KUKA KRL program: EPS_2_25252_PD3_A_20250910061716.src

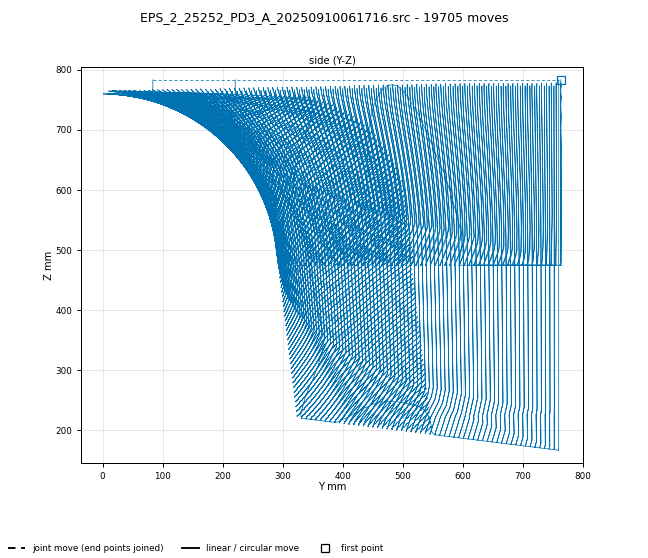
[picture p0: tool path of EPS_2_25252_PD3_A_20250910061716.src, 19705 of 19707 moves have a stored position in this frame; points joined in program order, loops and branches not executed]
&ACCESS RVP
&REL 4
&COMMENT QRS 19112012
&PARAM EDITMASK = *
DEF PART()
EXT BAS (BAS_COMMAND :IN,REAL :IN )
INT I
BAS (#INITMOV,0 )

;KUKA QRS Post kuka4.cps  Date:22-06-2017 !

File_ID=2831

QRS_PRE_INIT()

;Init var - Until changes are made in qrs_pre_init
Outlet_Square_prg=0
Inlet_1_Square_prg=0
Inlet_2_Square_prg=0
Inlet_3_Square_prg=0
Inlet_4_Square_prg=0
Inlet_5_Square_prg=0

Outlet_1={X 0.000, Y 612.000, Z 507.000, B 0.000, E1 0.000 }
Inlet_1={X 0.000, Y 651.000, Z 482.000, B 0.000, E1 180.000 }
Outlet_1_type=533
Inlet_1_type=0
;QRS#1=Sidecore dimensions
;QRS#2=525-21" Concrete
;QRS#3=DeadEnd 533
;QRS#4=
;QRS#5=
;QRS#6=
;QRS#7=
;QRS#8=
;QRS#9=S306-32
;QRS#10=

;QRS#11=
;QRS#12=
;QRS#13=
;QRS#14=
;QRS#15=
;QRS#16=1524x152x1219 4'
;QRS#17=EPS Height
;QRS#18=773,5
;QRS#19=*
;QRS#20= UPDATED VERSION 22-06-2017
;QRS#21=*
Outlet_Square=0350
Inlet_1_Square=00
Inlet_2_Square=0
Inlet_3_Square=0
Inlet_4_Square=0
Inlet_5_Square=0
Mill_Square=1
Outlet_Square_Prg=263
Inlet_1_Square_prg=0

QRS_INIT()

$ADVANCE=5

; T1
PTP {E1 176.574,E2 176.574}
PTP {X 0,Y 763.362,A -85,B 0,C 180,E1 176.574,E2 176.574,E3 0,E4 0,E5 0,E6 0}
QRS_SPEED_INIT()
LIN {X 0,Y 763.362,Z 783.5,A -85,B 0,C 180,E1 176.574,E2 176.574,E3 0,E4 0,E5 0,E6 0} C_VEL
LIN {X 0,Y 763.362,Z 476.78,A -85,B 0,C 180,E1 176.574,E2 176.574} C_VEL
LIN {X 0,Y 763.472,Z 474.78,A -85,B 0,C 180,E1 176.723,E2 176.723} C_VEL
LIN {X 0,Y 763.845,Z 474.78,A -85,B 0,C 180,E1 177.187,E2 177.187} C_VEL
LIN {X 0,Y 763.843,Z 474.78,A -85,B 0,C 180,E1 184.692,E2 184.692} C_VEL
LIN {X 0,Y 763.78,Z 474.78,A -85,B 0,C 180,E1 192.281,E2 192.281} C_VEL
LIN {X 0,Y 763.758,Z 474.78,A -85,B 0,C 180,E1 200.097,E2 200.097} C_VEL
LIN {X 0,Y 763.767,Z 474.78,A -85,B 0,C 180,E1 208.327,E2 208.327} C_VEL
LIN {X 0,Y 762.36,Z 474.78,A -85,B 0,C 180,E1 210.542,E2 210.542} C_VEL
LIN {X 0,Y 762.677,Z 474.78,A -85,B 0,C 180,E1 214.995,E2 214.995} C_VEL
LIN {X 0,Y 763.686,Z 474.78,A -85,B 0,C 180,E1 216.703,E2 216.703} C_VEL
LIN {X 0,Y 763.715,Z 474.78,A -85,B 0,C 180,E1 224.719,E2 224.719} C_VEL
LIN {X 0,Y 763.486,Z 474.78,A -85,B 0,C 180,E1 225.271,E2 225.271} C_VEL
LIN {X 0,Y 762.394,Z 474.78,A -85,B 0,C 180,E1 230.392,E2 230.392} C_VEL
LIN {X 0,Y 763.76,Z 474.78,A -85,B 0,C 180,E1 232.747,E2 232.747} C_VEL
LIN {X 0,Y 763.715,Z 474.78,A -85,B 0,C 180,E1 239.522,E2 239.522} C_VEL
LIN {X 0,Y 763.84,Z 474.78,A -85,B 0,C 180,E1 246.233,E2 246.233} C_VEL
LIN {X 0,Y 763.363,Z 474.78,A -85,B 0,C 180,E1 246.588,E2 246.588} C_VEL
LIN {X 0,Y 762.066,Z 474.78,A -85,B 0,C 180,E1 246.779,E2 246.779} C_VEL
LIN {X 0,Y 761.546,Z 474.78,A -85,B 0,C 180,E1 246.82,E2 246.82} C_VEL
LIN {X 0,Y 762.022,Z 475.377,A -85,B 0,C 180,E1 246.853,E2 246.853} C_VEL
LIN {X 0,Y 763.177,Z 477.146,A -85,B 0,C 180,E1 246.908,E2 246.908} C_VEL
LIN {X 0,Y 763.405,Z 477.716,A -85,B 0,C 180,E1 246.921,E2 246.921} C_VEL
LIN {X 0,Y 763.579,Z 479.406,A -85,B 0,C 180,E1 246.944,E2 246.944} C_VEL
LIN {X 0,Y 763.624,Z 506.616,A -85,B 0,C 180,E1 247.217,E2 247.217} C_VEL
LIN {X 0,Y 763.846,Z 526.018,A -85,B 0,C 180,E1 247.432,E2 247.432} C_VEL
LIN {X 0,Y 763.826,Z 535.654,A -85,B 0,C 180,E1 247.561,E2 247.561} C_VEL
LIN {X 0,Y 763.83,Z 546.762,A -85,B 0,C 180,E1 247.743,E2 247.743} C_VEL
LIN {X 0,Y 763.845,Z 560.557,A -85,B 0,C 180,E1 248.022,E2 248.022} C_VEL
LIN {X 0,Y 763.631,Z 572.226,A -85,B 0,C 180,E1 248.295,E2 248.295} C_VEL
LIN {X 0,Y 763.801,Z 585.949,A -85,B 0,C 180,E1 248.684,E2 248.684} C_VEL
LIN {X 0,Y 763.765,Z 598.566,A -85,B 0,C 180,E1 249.09,E2 249.09} C_VEL
LIN {X 0,Y 763.802,Z 611.561,A -85,B 0,C 180,E1 249.567,E2 249.567} C_VEL
LIN {X 0,Y 763.764,Z 623.559,A -85,B 0,C 180,E1 250.059,E2 250.059} C_VEL
LIN {X 0,Y 763.75,Z 634.569,A -85,B 0,C 180,E1 250.559,E2 250.559} C_VEL
LIN {X 0,Y 763.602,Z 646.52,A -85,B 0,C 180,E1 251.157,E2 251.157} C_VEL
LIN {X 0,Y 763.564,Z 657.079,A -85,B 0,C 180,E1 251.739,E2 251.739} C_VEL
LIN {X 0,Y 763.701,Z 667.628,A -85,B 0,C 180,E1 252.381,E2 252.381} C_VEL
LIN {X 0,Y 763.805,Z 676.976,A -85,B 0,C 180,E1 252.997,E2 252.997} C_VEL
LIN {X 0,Y 763.623,Z 687.198,A -85,B 0,C 180,E1 253.726,E2 253.726} C_VEL
LIN {X 0,Y 763.342,Z 695.759,A -85,B 0,C 180,E1 254.386,E2 254.386} C_VEL
LIN {X 0,Y 763.22,Z 704.692,A -85,B 0,C 180,E1 255.141,E2 255.141} C_VEL
LIN {X 0,Y 763.436,Z 713.229,A -85,B 0,C 180,E1 255.933,E2 255.933} C_VEL
LIN {X 0,Y 763.734,Z 720.481,A -85,B 0,C 180,E1 256.663,E2 256.663} C_VEL
LIN {X 0,Y 763.713,Z 726.434,A -85,B 0,C 180,E1 257.312,E2 257.312} C_VEL
LIN {X 0,Y 763.274,Z 733.979,A -85,B 0,C 180,E1 258.192,E2 258.192} C_VEL
LIN {X 0,Y 763.073,Z 741.325,A -85,B 0,C 180,E1 259.146,E2 259.146} C_VEL
LIN {X 0,Y 763.305,Z 747.875,A -85,B 0,C 180,E1 260.102,E2 260.102} C_VEL
LIN {X 0,Y 763.778,Z 753.687,A -85,B 0,C 180,E1 261.059,E2 261.059} C_VEL
LIN {X 0,Y 763.865,Z 755,A -85,B 0,C 180,E1 261.297,E2 261.297} C_VEL
LIN {X 0,Y 763.317,Z 759.964,A -85,B 0,C 180,E1 262.238,E2 262.238} C_VEL
LIN {X 0,Y 762.989,Z 763.277,A -85,B 0,C 180,E1 262.945,E2 262.945} C_VEL
LIN {X 0,Y 762.889,Z 767.126,A -85,B 0,C 180,E1 263.888,E2 263.888} C_VEL
LIN {X 0,Y 763.222,Z 770.376,A -85,B 0,C 180,E1 264.834,E2 264.834} C_VEL
LIN {X 0,Y 763.816,Z 773.348,A -85,B 0,C 180,E1 265.894,E2 265.894} C_VEL
LIN {X 0,Y 763.592,Z 774.667,A -85,B 0,C 180,E1 266.478,E2 266.478} C_VEL
LIN {X 0,Y 763.145,Z 776.072,A -85,B 0,C 180,E1 267.184,E2 267.184} C_VEL
LIN {X 0,Y 762.829,Z 777.16,A -85,B 0,C 180,E1 267.91,E2 267.91} C_VEL
LIN {X 0,Y 762.834,Z 778.22,A -85,B 0,C 180,E1 269.061,E2 269.061} C_VEL
LIN {X 0,Y 763.862,Z 778.174,A -85,B 0,C 180,E1 270.937,E2 270.937} C_VEL
LIN {X 0,Y 763.613,Z 777.551,A -85,B 0,C 180,E1 271.688,E2 271.688} C_VEL
LIN {X 0,Y 763.495,Z 776.058,A -85,B 0,C 180,E1 272.814,E2 272.814} C_VEL
LIN {X 0,Y 763.659,Z 774.541,A -85,B 0,C 180,E1 273.58,E2 273.58} C_VEL
LIN {X 0,Y 763.841,Z 773.267,A -85,B 0,C 180,E1 274.135,E2 274.135} C_VEL
LIN {X 0,Y 763.624,Z 771.764,A -85,B 0,C 180,E1 274.693,E2 274.693} C_VEL
LIN {X 0,Y 763.089,Z 768.798,A -85,B 0,C 180,E1 275.638,E2 275.638} C_VEL
LIN {X 0,Y 762.918,Z 767.126,A -85,B 0,C 180,E1 276.111,E2 276.111} C_VEL
LIN {X 0,Y 762.9,Z 763.277,A -85,B 0,C 180,E1 277.056,E2 277.056} C_VEL
LIN {X 0,Y 763.306,Z 758.808,A -85,B 0,C 180,E1 277.998,E2 277.998} C_VEL
LIN {X 0,Y 763.85,Z 753.687,A -85,B 0,C 180,E1 278.94,E2 278.94} C_VEL
LIN {X 0,Y 763.421,Z 747.875,A -85,B 0,C 180,E1 279.896,E2 279.896} C_VEL
LIN {X 0,Y 763.086,Z 741.325,A -85,B 0,C 180,E1 280.854,E2 280.854} C_VEL
LIN {X 0,Y 763.195,Z 733.979,A -85,B 0,C 180,E1 281.809,E2 281.809} C_VEL
LIN {X 0,Y 763.537,Z 727.593,A -85,B 0,C 180,E1 282.565,E2 282.565} C_VEL
LIN {X 0,Y 763.83,Z 720.63,A -85,B 0,C 180,E1 283.319,E2 283.319} C_VEL
LIN {X 0,Y 763.441,Z 710.557,A -85,B 0,C 180,E1 284.319,E2 284.319} C_VEL
LIN {X 0,Y 763.239,Z 702.208,A -85,B 0,C 180,E1 285.074,E2 285.074} C_VEL
LIN {X 0,Y 763.3,Z 694.06,A -85,B 0,C 180,E1 285.751,E2 285.751} C_VEL
LIN {X 0,Y 763.618,Z 683.872,A -85,B 0,C 180,E1 286.518,E2 286.518} C_VEL
LIN {X 0,Y 763.769,Z 675.166,A -85,B 0,C 180,E1 287.127,E2 287.127} C_VEL
LIN {X 0,Y 763.695,Z 663.646,A -85,B 0,C 180,E1 287.866,E2 287.866} C_VEL
LIN {X 0,Y 763.565,Z 654.622,A -85,B 0,C 180,E1 288.403,E2 288.403} C_VEL
LIN {X 0,Y 763.593,Z 642.535,A -85,B 0,C 180,E1 289.05,E2 289.05} C_VEL
LIN {X 0,Y 763.737,Z 630.359,A -85,B 0,C 180,E1 289.637,E2 289.637} C_VEL
LIN {X 0,Y 763.711,Z 620.01,A -85,B 0,C 180,E1 290.096,E2 290.096} C_VEL
LIN {X 0,Y 763.808,Z 608.143,A -85,B 0,C 180,E1 290.566,E2 290.566} C_VEL
LIN {X 0,Y 763.711,Z 594.677,A -85,B 0,C 180,E1 291.043,E2 291.043} C_VEL
LIN {X 0,Y 763.729,Z 582.345,A -85,B 0,C 180,E1 291.425,E2 291.425} C_VEL
LIN {X 0,Y 763.792,Z 568.153,A -85,B 0,C 180,E1 291.801,E2 291.801} C_VEL
LIN {X 0,Y 763.649,Z 556.327,A -85,B 0,C 180,E1 292.077,E2 292.077} C_VEL
LIN {X 0,Y 763.845,Z 541.803,A -85,B 0,C 180,E1 292.342,E2 292.342} C_VEL
LIN {X 0,Y 763.851,Z 529.818,A -85,B 0,C 180,E1 292.523,E2 292.523} C_VEL
LIN {X 0,Y 763.83,Z 511.799,A -85,B 0,C 180,E1 292.724,E2 292.724} C_VEL
LIN {X 0,Y 763.611,Z 481.566,A -85,B 0,C 180,E1 293.034,E2 293.034} C_VEL
LIN {X 0,Y 763.361,Z 477.535,A -85,B 0,C 180,E1 293.082,E2 293.082} C_VEL
LIN {X 0,Y 762.558,Z 474.78,A -85,B 0,C 180,E1 293.148,E2 293.148} C_VEL
LIN {X 0,Y 763.365,Z 474.78,A -85,B 0,C 180,E1 293.244,E2 293.244} C_VEL
LIN {X 0,Y 763.723,Z 474.78,A -85,B 0,C 180,E1 293.756,E2 293.756} C_VEL
LIN {X 0,Y 763.844,Z 474.78,A -85,B 0,C 180,E1 298.32,E2 298.32} C_VEL
LIN {X 0,Y 763.726,Z 474.78,A -85,B 0,C 180,E1 304.935,E2 304.935} C_VEL
LIN {X 0,Y 762.49,Z 474.78,A -85,B 0,C 180,E1 307.326,E2 307.326} C_VEL
LIN {X 0,Y 763.687,Z 474.78,A -85,B 0,C 180,E1 312.132,E2 312.132} C_VEL
LIN {X 0,Y 763.532,Z 474.78,A -85,B 0,C 180,E1 312.563,E2 312.563} C_VEL
LIN {X 0,Y 763.766,Z 474.78,A -85,B 0,C 180,E1 320.258,E2 320.258} C_VEL
LIN {X 0,Y 763.66,Z 474.78,A -85,B 0,C 180,E1 326.563,E2 326.563} C_VEL
LIN {X 0,Y 763.416,Z 474.78,A -85,B 0,C 180,E1 327.302,E2 327.302} C_VEL
LIN {X 0,Y 763.767,Z 474.78,A -85,B 0,C 180,E1 333.782,E2 333.782} C_VEL
LIN {X 0,Y 763.76,Z 474.78,A -85,B 0,C 180,E1 341.887,E2 341.887} C_VEL
LIN {X 0,Y 763.788,Z 474.78,A -85,B 0,C 180,E1 349.631,E2 349.631} C_VEL
LIN {X 0,Y 763.844,Z 474.78,A -85,B 0,C 180,E1 357.187,E2 357.187} C_VEL
LIN {X 0,Y 763.835,Z 474.78,A -85,B 0,C 180,E1 364.692,E2 364.692} C_VEL
LIN {X 0,Y 763.773,Z 474.78,A -85,B 0,C 180,E1 372.281,E2 372.281} C_VEL
LIN {X 0,Y 763.757,Z 474.78,A -85,B 0,C 180,E1 380.097,E2 380.097} C_VEL
LIN {X 0,Y 763.776,Z 474.78,A -85,B 0,C 180,E1 388.327,E2 388.327} C_VEL
LIN {X 0,Y 763.753,Z 474.78,A -85,B 0,C 180,E1 394.938,E2 394.938} C_VEL
LIN {X 0,Y 762.455,Z 474.78,A -85,B 0,C 180,E1 399.735,E2 399.735} C_VEL
LIN {X 0,Y 763.747,Z 474.78,A -85,B 0,C 180,E1 402.135,E2 402.135} C_VEL
LIN {X 0,Y 763.573,Z 474.78,A -85,B 0,C 180,E1 402.574,E2 402.574} C_VEL
LIN {X 0,Y 763.844,Z 474.78,A -85,B 0,C 180,E1 410.26,E2 410.26} C_VEL
LIN {X 0,Y 763.674,Z 474.78,A -85,B 0,C 180,E1 416.573,E2 416.573} C_VEL
LIN {X 0,Y 763.421,Z 474.78,A -85,B 0,C 180,E1 417.307,E2 417.307} C_VEL
LIN {X 0,Y 763.747,Z 474.78,A -85,B 0,C 180,E1 423.785,E2 423.785} C_VEL
LIN {X 0,Y 763.796,Z 474.78,A -85,B 0,C 180,E1 431.89,E2 431.89} C_VEL
LIN {X 0,Y 763.784,Z 474.78,A -85,B 0,C 180,E1 439.633,E2 439.633} C_VEL
LIN {X 0,Y 763.772,Z 474.78,A -85,B 0,C 180,E1 447.187,E2 447.187} C_VEL
LIN {X 0,Y 763.776,Z 474.78,A -85,B 0,C 180,E1 454.692,E2 454.692} C_VEL
LIN {X 0,Y 763.786,Z 474.78,A -85,B 0,C 180,E1 462.279,E2 462.279} C_VEL
LIN {X 0,Y 763.785,Z 474.78,A -85,B 0,C 180,E1 470.094,E2 470.094} C_VEL
LIN {X 0,Y 763.728,Z 474.78,A -85,B 0,C 180,E1 478.325,E2 478.325} C_VEL
LIN {X 0,Y 761.89,Z 474.78,A -85,B 0,C 180,E1 482.767,E2 482.767} C_VEL
LIN {X 0,Y 762.616,Z 474.78,A -85,B 0,C 180,E1 484.993,E2 484.993} C_VEL
LIN {X 0,Y 763.623,Z 474.78,A -85,B 0,C 180,E1 486.687,E2 486.687} C_VEL
LIN {X 0,Y 763.669,Z 474.78,A -85,B 0,C 180,E1 494.715,E2 494.715} C_VEL
LIN {X 0,Y 763.456,Z 474.78,A -85,B 0,C 180,E1 495.262,E2 495.262} C_VEL
LIN {X 0,Y 762.344,Z 474.78,A -85,B 0,C 180,E1 500.387,E2 500.387} C_VEL
LIN {X 0,Y 763.704,Z 474.78,A -85,B 0,C 180,E1 502.738,E2 502.738} C_VEL
LIN {X 0,Y 763.588,Z 474.78,A -85,B 0,C 180,E1 510.146,E2 510.146} C_VEL
LIN {X 0,Y 762.882,Z 474.78,A -85,B 0,C 180,E1 511.637,E2 511.637} C_VEL
LIN {X 0,Y 763.752,Z 474.78,A -85,B 0,C 180,E1 517.893,E2 517.893} C_VEL
LIN {X 0,Y 763.489,Z 474.78,A -85,B 0,C 180,E1 524.93,E2 524.93} C_VEL
LIN {X 0,Y 763.662,Z 474.78,A -85,B 0,C 180,E1 525.79,E2 525.79} C_VEL
LIN {X 0,Y 763.795,Z 474.78,A -85,B 0,C 180,E1 529.631,E2 529.631} C_VEL
LIN {X 0,Y 763.472,Z 474.78,A -85,B 0,C 180,E1 536.723,E2 536.723} C_VEL
LIN {X 0,Y 754.509,Z 474.78,A -85,B 0,C 180,E1 539.325,E2 539.325} C_VEL
LIN {X 0,Y 754.692,Z 474.78,A -85,B 0,C 180,E1 546.383,E2 546.383} C_VEL
LIN {X 0,Y 754.905,Z 474.78,A -85,B 0,C 180,E1 553.399,E2 553.399} C_VEL
LIN {X 0,Y 755.041,Z 474.78,A -85,B 0,C 180,E1 560.942,E2 560.942} C_VEL
LIN {X 0,Y 754.868,Z 474.78,A -85,B 0,C 180,E1 569.54,E2 569.54} C_VEL
LIN {X 0,Y 754.766,Z 474.78,A -85,B 0,C 180,E1 577.858,E2 577.858} C_VEL
LIN {X 0,Y 754.887,Z 474.78,A -85,B 0,C 180,E1 586.126,E2 586.126} C_VEL
LIN {X 0,Y 755.149,Z 474.78,A -85,B 0,C 180,E1 593.671,E2 593.671} C_VEL
LIN {X 0,Y 754.823,Z 474.78,A -85,B 0,C 180,E1 601.041,E2 601.041} C_VEL
LIN {X 0,Y 754.166,Z 474.78,A -85,B 0,C 180,E1 606.591,E2 606.591} C_VEL
LIN {X 0,Y 756.39,Z 562.55,A -85,B 0,C 180,E1 607.841,E2 607.841} C_VEL
LIN {X 0,Y 756.168,Z 623.267,A -85,B 0,C 180,E1 609.837,E2 609.837} C_VEL
LIN {X 0,Y 756.007,Z 677.473,A -85,B 0,C 180,E1 612.852,E2 612.852} C_VEL
LIN {X 0,Y 755.802,Z 721.742,A -85,B 0,C 180,E1 616.659,E2 616.659} C_VEL
LIN {X 0,Y 755.794,Z 754.21,A -85,B 0,C 180,E1 621.054,E2 621.054} C_VEL
LIN {X 0,Y 755.805,Z 773.709,A -85,B 0,C 180,E1 625.973,E2 625.973} C_VEL
LIN {X 0,Y 755.615,Z 778.34,A -85,B 0,C 180,E1 630.575,E2 630.575} C_VEL
LIN {X 0,Y 755.326,Z 770.506,A -85,B 0,C 180,E1 635.184,E2 635.184} C_VEL
LIN {X 0,Y 755.484,Z 748.988,A -85,B 0,C 180,E1 639.824,E2 639.824} C_VEL
LIN {X 0,Y 755.589,Z 713.063,A -85,B 0,C 180,E1 644.233,E2 644.233} C_VEL
LIN {X 0,Y 755.936,Z 664.27,A -85,B 0,C 180,E1 648.018,E2 648.018} C_VEL
LIN {X 0,Y 756.249,Z 606.531,A -85,B 0,C 180,E1 650.84,E2 650.84} C_VEL
LIN {X 0,Y 756.434,Z 543.515,A -85,B 0,C 180,E1 652.545,E2 652.545} C_VEL
LIN {X 0,Y 755.352,Z 474.78,A -85,B 0,C 180,E1 653.409,E2 653.409} C_VEL
LIN {X 0,Y 755.098,Z 474.78,A -85,B 0,C 180,E1 659.475,E2 659.475} C_VEL
LIN {X 0,Y 754.862,Z 474.78,A -85,B 0,C 180,E1 666.345,E2 666.345} C_VEL
LIN {X 0,Y 755.342,Z 474.78,A -85,B 0,C 180,E1 672.798,E2 672.798} C_VEL
LIN {X 0,Y 755.448,Z 474.78,A -85,B 0,C 180,E1 680.711,E2 680.711} C_VEL
LIN {X 0,Y 755.103,Z 474.78,A -85,B 0,C 180,E1 687.787,E2 687.787} C_VEL
LIN {X 0,Y 755.266,Z 474.78,A -85,B 0,C 180,E1 694.373,E2 694.373} C_VEL
LIN {X 0,Y 754.891,Z 474.78,A -85,B 0,C 180,E1 703.021,E2 703.021} C_VEL
LIN {X 0,Y 755.374,Z 474.78,A -85,B 0,C 180,E1 710.135,E2 710.135} C_VEL
LIN {X 0,Y 755.05,Z 474.78,A -85,B 0,C 180,E1 718.238,E2 718.238} C_VEL
LIN {X 0,Y 754.845,Z 474.78,A -85,B 0,C 180,E1 726.036,E2 726.036} C_VEL
LIN {X 0,Y 754.937,Z 474.78,A -85,B 0,C 180,E1 733.327,E2 733.327} C_VEL
LIN {X 0,Y 755.046,Z 474.78,A -85,B 0,C 180,E1 740.943,E2 740.943} C_VEL
LIN {X 0,Y 755.058,Z 474.78,A -85,B 0,C 180,E1 749.452,E2 749.452} C_VEL
LIN {X 0,Y 754.823,Z 474.78,A -85,B 0,C 180,E1 756.324,E2 756.324} C_VEL
LIN {X 0,Y 755.323,Z 474.78,A -85,B 0,C 180,E1 762.877,E2 762.877} C_VEL
LIN {X 0,Y 755.472,Z 474.78,A -85,B 0,C 180,E1 770.779,E2 770.779} C_VEL
LIN {X 0,Y 755.079,Z 474.78,A -85,B 0,C 180,E1 777.844,E2 777.844} C_VEL
LIN {X 0,Y 755.203,Z 474.78,A -85,B 0,C 180,E1 784.423,E2 784.423} C_VEL
LIN {X 0,Y 754.891,Z 474.78,A -85,B 0,C 180,E1 793.065,E2 793.065} C_VEL
LIN {X 0,Y 755.331,Z 474.78,A -85,B 0,C 180,E1 800.174,E2 800.174} C_VEL
LIN {X 0,Y 754.958,Z 474.78,A -85,B 0,C 180,E1 808.273,E2 808.273} C_VEL
LIN {X 0,Y 754.788,Z 474.78,A -85,B 0,C 180,E1 816.063,E2 816.063} C_VEL
LIN {X 0,Y 754.932,Z 474.78,A -85,B 0,C 180,E1 823.357,E2 823.357} C_VEL
LIN {X 0,Y 755.023,Z 474.78,A -85,B 0,C 180,E1 830.963,E2 830.963} C_VEL
LIN {X 0,Y 754.794,Z 474.78,A -85,B 0,C 180,E1 839.488,E2 839.488} C_VEL
LIN {X 0,Y 754.728,Z 474.78,A -85,B 0,C 180,E1 847.795,E2 847.795} C_VEL
LIN {X 0,Y 754.835,Z 474.78,A -85,B 0,C 180,E1 856.144,E2 856.144} C_VEL
LIN {X 0,Y 754.97,Z 474.78,A -85,B 0,C 180,E1 863.684,E2 863.684} C_VEL
LIN {X 0,Y 754.771,Z 474.78,A -85,B 0,C 180,E1 871.85,E2 871.85} C_VEL
LIN {X 0,Y 754.717,Z 474.78,A -85,B 0,C 180,E1 879.439,E2 879.439} C_VEL
LIN {X 0,Y 755.375,Z 474.78,A -85,B 0,C 180,E1 886.827,E2 886.827} C_VEL
LIN {X 0,Y 754.178,Z 474.78,A -85,B 0,C 180,E1 893.682,E2 893.682} C_VEL
LIN {X 0,Y 755.031,Z 474.78,A -85,B 0,C 180,E1 898.307,E2 898.307} C_VEL
LIN {X 0,Y 754.509,Z 474.78,A -85,B 0,C 180,E1 899.325,E2 899.325} C_VEL
LIN {X 0,Y 746.359,Z 474.78,A -85,B 0,C 180,E1 901.958,E2 901.958} C_VEL
LIN {X 0,Y 746.234,Z 474.78,A -85,B 0,C 180,E1 907.629,E2 907.629} C_VEL
LIN {X 0,Y 746.807,Z 474.78,A -85,B 0,C 180,E1 913.547,E2 913.547} C_VEL
LIN {X 0,Y 747.111,Z 474.78,A -85,B 0,C 180,E1 920.854,E2 920.854} C_VEL
LIN {X 0,Y 747.442,Z 474.78,A -85,B 0,C 180,E1 928.531,E2 928.531} C_VEL
LIN {X 0,Y 747.23,Z 474.78,A -85,B 0,C 180,E1 936.841,E2 936.841} C_VEL
LIN {X 0,Y 747.247,Z 474.78,A -85,B 0,C 180,E1 945.561,E2 945.561} C_VEL
LIN {X 0,Y 747.244,Z 474.78,A -85,B 0,C 180,E1 953.381,E2 953.381} C_VEL
LIN {X 0,Y 747.137,Z 474.78,A -85,B 0,C 180,E1 960.179,E2 960.179} C_VEL
LIN {X 0,Y 746.841,Z 475.472,A -85,B 0,C 180,E1 966.356,E2 966.356} C_VEL
LIN {X 0,Y 748.969,Z 562.274,A -85,B 0,C 180,E1 967.603,E2 967.603} C_VEL
LIN {X 0,Y 748.558,Z 623.266,A -85,B 0,C 180,E1 969.623,E2 969.623} C_VEL
LIN {X 0,Y 748.205,Z 677.856,A -85,B 0,C 180,E1 972.695,E2 972.695} C_VEL
LIN {X 0,Y 747.901,Z 723.112,A -85,B 0,C 180,E1 976.669,E2 976.669} C_VEL
LIN {X 0,Y 747.831,Z 755.753,A -85,B 0,C 180,E1 981.252,E2 981.252} C_VEL
LIN {X 0,Y 747.79,Z 773.708,A -85,B 0,C 180,E1 985.93,E2 985.93} C_VEL
LIN {X 0,Y 747.609,Z 778.34,A -85,B 0,C 180,E1 990.581,E2 990.581} C_VEL
LIN {X 0,Y 747.293,Z 770.508,A -85,B 0,C 180,E1 995.239,E2 995.239} C_VEL
LIN {X 0,Y 747.479,Z 748.984,A -85,B 0,C 180,E1 999.93,E2 999.93} C_VEL
LIN {X 0,Y 747.658,Z 713.056,A -85,B 0,C 180,E1 1004.387,E2 1004.387} C_VEL
LIN {X 0,Y 748.186,Z 664.011,A -85,B 0,C 180,E1 1008.227,E2 1008.227} C_VEL
LIN {X 0,Y 748.669,Z 606.542,A -85,B 0,C 180,E1 1011.061,E2 1011.061} C_VEL
LIN {X 0,Y 749.031,Z 544.136,A -85,B 0,C 180,E1 1012.769,E2 1012.769} C_VEL
LIN {X 0,Y 747.589,Z 474.78,A -85,B 0,C 180,E1 1013.718,E2 1013.718} C_VEL
LIN {X 0,Y 746.777,Z 474.78,A -85,B 0,C 180,E1 1020.223,E2 1020.223} C_VEL
LIN {X 0,Y 746.686,Z 474.78,A -85,B 0,C 180,E1 1026.808,E2 1026.808} C_VEL
LIN {X 0,Y 746.669,Z 474.78,A -85,B 0,C 180,E1 1033.783,E2 1033.783} C_VEL
LIN {X 0,Y 746.949,Z 474.78,A -85,B 0,C 180,E1 1041.674,E2 1041.674} C_VEL
LIN {X 0,Y 746.669,Z 474.78,A -85,B 0,C 180,E1 1048.751,E2 1048.751} C_VEL
LIN {X 0,Y 746.571,Z 474.78,A -85,B 0,C 180,E1 1055.341,E2 1055.341} C_VEL
LIN {X 0,Y 747.02,Z 474.78,A -85,B 0,C 180,E1 1062.836,E2 1062.836} C_VEL
LIN {X 0,Y 746.698,Z 474.78,A -85,B 0,C 180,E1 1071.199,E2 1071.199} C_VEL
LIN {X 0,Y 747.053,Z 474.78,A -85,B 0,C 180,E1 1078.219,E2 1078.219} C_VEL
LIN {X 0,Y 747.412,Z 474.78,A -85,B 0,C 180,E1 1085.206,E2 1085.206} C_VEL
LIN {X 0,Y 746.837,Z 474.78,A -85,B 0,C 180,E1 1093.475,E2 1093.475} C_VEL
LIN {X 0,Y 747.157,Z 474.78,A -85,B 0,C 180,E1 1100.778,E2 1100.778} C_VEL
LIN {X 0,Y 747.444,Z 474.78,A -85,B 0,C 180,E1 1108.451,E2 1108.451} C_VEL
LIN {X 0,Y 747.436,Z 474.78,A -85,B 0,C 180,E1 1115.304,E2 1115.304} C_VEL
LIN {X 0,Y 747.357,Z 474.78,A -85,B 0,C 180,E1 1122.803,E2 1122.803} C_VEL
LIN {X 0,Y 746.965,Z 474.78,A -85,B 0,C 180,E1 1131.742,E2 1131.742} C_VEL
LIN {X 0,Y 746.637,Z 474.78,A -85,B 0,C 180,E1 1138.807,E2 1138.807} C_VEL
LIN {X 0,Y 746.534,Z 474.78,A -85,B 0,C 180,E1 1145.391,E2 1145.391} C_VEL
LIN {X 0,Y 747.005,Z 474.78,A -85,B 0,C 180,E1 1152.881,E2 1152.881} C_VEL
LIN {X 0,Y 747.314,Z 474.78,A -85,B 0,C 180,E1 1160.068,E2 1160.068} C_VEL
LIN {X 0,Y 746.961,Z 474.78,A -85,B 0,C 180,E1 1168.255,E2 1168.255} C_VEL
LIN {X 0,Y 747.336,Z 474.78,A -85,B 0,C 180,E1 1175.239,E2 1175.239} C_VEL
LIN {X 0,Y 746.833,Z 474.78,A -85,B 0,C 180,E1 1183.504,E2 1183.504} C_VEL
LIN {X 0,Y 747.137,Z 474.78,A -85,B 0,C 180,E1 1190.806,E2 1190.806} C_VEL
LIN {X 0,Y 747.373,Z 474.78,A -85,B 0,C 180,E1 1198.479,E2 1198.479} C_VEL
LIN {X 0,Y 747.147,Z 474.78,A -85,B 0,C 180,E1 1206.781,E2 1206.781} C_VEL
LIN {X 0,Y 746.84,Z 474.78,A -85,B 0,C 180,E1 1216.124,E2 1216.124} C_VEL
LIN {X 0,Y 747.112,Z 474.78,A -85,B 0,C 180,E1 1223.3,E2 1223.3} C_VEL
LIN {X 0,Y 746.661,Z 474.78,A -85,B 0,C 180,E1 1232.067,E2 1232.067} C_VEL
LIN {X 0,Y 746.852,Z 474.78,A -85,B 0,C 180,E1 1239.213,E2 1239.213} C_VEL
LIN {X 0,Y 747.328,Z 474.78,A -85,B 0,C 180,E1 1247.728,E2 1247.728} C_VEL
LIN {X 0,Y 747.783,Z 474.78,A -85,B 0,C 180,E1 1257.127,E2 1257.127} C_VEL
LIN {X 0,Y 746.359,Z 474.78,A -85,B 0,C 180,E1 1261.958,E2 1261.958} C_VEL
LIN {X 0,Y 739.299,Z 474.78,A -85,B 0,C 180,E1 1264.638,E2 1264.638} C_VEL
LIN {X 0,Y 738.728,Z 474.78,A -85,B 0,C 180,E1 1273.698,E2 1273.698} C_VEL
LIN {X 0,Y 738.919,Z 474.78,A -85,B 0,C 180,E1 1281.097,E2 1281.097} C_VEL
LIN {X 0,Y 738.946,Z 474.78,A -85,B 0,C 180,E1 1289.285,E2 1289.285} C_VEL
LIN {X 0,Y 738.703,Z 474.78,A -85,B 0,C 180,E1 1297.78,E2 1297.78} C_VEL
LIN {X 0,Y 739.312,Z 474.78,A -85,B 0,C 180,E1 1305.123,E2 1305.123} C_VEL
LIN {X 0,Y 738.84,Z 474.78,A -85,B 0,C 180,E1 1314.267,E2 1314.267} C_VEL
LIN {X 0,Y 738.752,Z 474.78,A -85,B 0,C 180,E1 1321.158,E2 1321.158} C_VEL
LIN {X 0,Y 739.506,Z 476.426,A -85,B 0,C 180,E1 1326.116,E2 1326.116} C_VEL
LIN {X 0,Y 741.559,Z 562.703,A -85,B 0,C 180,E1 1327.377,E2 1327.377} C_VEL
LIN {X 0,Y 740.98,Z 623.251,A -85,B 0,C 180,E1 1329.405,E2 1329.405} C_VEL
LIN {X 0,Y 740.408,Z 678.774,A -85,B 0,C 180,E1 1332.575,E2 1332.575} C_VEL
LIN {X 0,Y 739.988,Z 723.549,A -85,B 0,C 180,E1 1336.573,E2 1336.573} C_VEL
LIN {X 0,Y 739.826,Z 755.755,A -85,B 0,C 180,E1 1341.157,E2 1341.157} C_VEL
LIN {X 0,Y 739.762,Z 773.706,A -85,B 0,C 180,E1 1345.886,E2 1345.886} C_VEL
LIN {X 0,Y 739.603,Z 778.34,A -85,B 0,C 180,E1 1350.587,E2 1350.587} C_VEL
LIN {X 0,Y 739.288,Z 770.51,A -85,B 0,C 180,E1 1355.296,E2 1355.296} C_VEL
LIN {X 0,Y 739.489,Z 748.981,A -85,B 0,C 180,E1 1360.039,E2 1360.039} C_VEL
LIN {X 0,Y 739.734,Z 713.05,A -85,B 0,C 180,E1 1364.544,E2 1364.544} C_VEL
LIN {X 0,Y 740.441,Z 664.852,A -85,B 0,C 180,E1 1368.372,E2 1368.372} C_VEL
LIN {X 0,Y 741.129,Z 606.769,A -85,B 0,C 180,E1 1371.277,E2 1371.277} C_VEL
LIN {X 0,Y 741.675,Z 542.984,A -85,B 0,C 180,E1 1373.027,E2 1373.027} C_VEL
LIN {X 0,Y 739.593,Z 474.78,A -85,B 0,C 180,E1 1373.917,E2 1373.917} C_VEL
LIN {X 0,Y 738.533,Z 474.78,A -85,B 0,C 180,E1 1381.441,E2 1381.441} C_VEL
LIN {X 0,Y 738.412,Z 474.78,A -85,B 0,C 180,E1 1387.658,E2 1387.658} C_VEL
LIN {X 0,Y 738.865,Z 474.78,A -85,B 0,C 180,E1 1393.438,E2 1393.438} C_VEL
LIN {X 0,Y 739.098,Z 474.78,A -85,B 0,C 180,E1 1401.192,E2 1401.192} C_VEL
LIN {X 0,Y 738.801,Z 474.78,A -85,B 0,C 180,E1 1408.413,E2 1408.413} C_VEL
LIN {X 0,Y 738.763,Z 474.78,A -85,B 0,C 180,E1 1415.063,E2 1415.063} C_VEL
LIN {X 0,Y 739.103,Z 474.78,A -85,B 0,C 180,E1 1422.646,E2 1422.646} C_VEL
LIN {X 0,Y 738.736,Z 474.78,A -85,B 0,C 180,E1 1431.104,E2 1431.104} C_VEL
LIN {X 0,Y 739.057,Z 474.78,A -85,B 0,C 180,E1 1438.2,E2 1438.2} C_VEL
LIN {X 0,Y 739.091,Z 474.78,A -85,B 0,C 180,E1 1445.654,E2 1445.654} C_VEL
LIN {X 0,Y 738.764,Z 474.78,A -85,B 0,C 180,E1 1453.625,E2 1453.625} C_VEL
LIN {X 0,Y 738.989,Z 474.78,A -85,B 0,C 180,E1 1461.019,E2 1461.019} C_VEL
LIN {X 0,Y 739.049,Z 474.78,A -85,B 0,C 180,E1 1469.299,E2 1469.299} C_VEL
LIN {X 0,Y 739.064,Z 474.78,A -85,B 0,C 180,E1 1475.855,E2 1475.855} C_VEL
LIN {X 0,Y 738.916,Z 474.78,A -85,B 0,C 180,E1 1483.412,E2 1483.412} C_VEL
LIN {X 0,Y 739.18,Z 474.78,A -85,B 0,C 180,E1 1491.264,E2 1491.264} C_VEL
LIN {X 0,Y 738.751,Z 474.78,A -85,B 0,C 180,E1 1498.436,E2 1498.436} C_VEL
LIN {X 0,Y 738.7,Z 474.78,A -85,B 0,C 180,E1 1505.112,E2 1505.112} C_VEL
LIN {X 0,Y 739.073,Z 474.78,A -85,B 0,C 180,E1 1512.691,E2 1512.691} C_VEL
LIN {X 0,Y 738.739,Z 474.78,A -85,B 0,C 180,E1 1521.144,E2 1521.144} C_VEL
LIN {X 0,Y 738.965,Z 474.78,A -85,B 0,C 180,E1 1528.236,E2 1528.236} C_VEL
LIN {X 0,Y 739.026,Z 474.78,A -85,B 0,C 180,E1 1535.683,E2 1535.683} C_VEL
LIN {X 0,Y 738.761,Z 474.78,A -85,B 0,C 180,E1 1543.654,E2 1543.654} C_VEL
LIN {X 0,Y 738.952,Z 474.78,A -85,B 0,C 180,E1 1551.047,E2 1551.047} C_VEL
LIN {X 0,Y 738.858,Z 474.78,A -85,B 0,C 180,E1 1559.296,E2 1559.296} C_VEL
LIN {X 0,Y 738.618,Z 474.78,A -85,B 0,C 180,E1 1567.794,E2 1567.794} C_VEL
LIN {X 0,Y 739.273,Z 474.78,A -85,B 0,C 180,E1 1575.049,E2 1575.049} C_VEL
LIN {X 0,Y 738.627,Z 474.78,A -85,B 0,C 180,E1 1584.211,E2 1584.211} C_VEL
LIN {X 0,Y 738.924,Z 474.78,A -85,B 0,C 180,E1 1591.19,E2 1591.19} C_VEL
LIN {X 0,Y 738.923,Z 474.78,A -85,B 0,C 180,E1 1599.034,E2 1599.034} C_VEL
LIN {X 0,Y 739.32,Z 474.78,A -85,B 0,C 180,E1 1607.592,E2 1607.592} C_VEL
LIN {X 0,Y 739.742,Z 474.78,A -85,B 0,C 180,E1 1617.096,E2 1617.096} C_VEL
LIN {X 0,Y 739.299,Z 474.78,A -85,B 0,C 180,E1 1624.638,E2 1624.638} C_VEL
LIN {X 0,Y 730.319,Z 474.78,A -85,B 0,C 180,E1 1627.314,E2 1627.314} C_VEL
LIN {X 0,Y 730.642,Z 474.78,A -85,B 0,C 180,E1 1633.853,E2 1633.853} C_VEL
LIN {X 0,Y 730.744,Z 474.78,A -85,B 0,C 180,E1 1641.344,E2 1641.344} C_VEL
LIN {X 0,Y 730.968,Z 474.78,A -85,B 0,C 180,E1 1649.235,E2 1649.235} C_VEL
LIN {X 0,Y 730.687,Z 474.78,A -85,B 0,C 180,E1 1657.819,E2 1657.819} C_VEL
LIN {X 0,Y 730.867,Z 474.78,A -85,B 0,C 180,E1 1665.965,E2 1665.965} C_VEL
LIN {X 0,Y 730.903,Z 474.78,A -85,B 0,C 180,E1 1673.749,E2 1673.749} C_VEL
LIN {X 0,Y 730.898,Z 474.78,A -85,B 0,C 180,E1 1680.818,E2 1680.818} C_VEL
LIN {X 0,Y 731.284,Z 475.314,A -85,B 0,C 180,E1 1685.819,E2 1685.819} C_VEL
LIN {X 0,Y 734.249,Z 506.523,A -85,B 0,C 180,E1 1686.25,E2 1686.25} C_VEL
LIN {X 0,Y 733.85,Z 574.284,A -85,B 0,C 180,E1 1687.426,E2 1687.426} C_VEL
LIN {X 0,Y 733.236,Z 634.845,A -85,B 0,C 180,E1 1689.731,E2 1689.731} C_VEL
LIN {X 0,Y 732.474,Z 686.979,A -85,B 0,C 180,E1 1692.996,E2 1692.996} C_VEL
LIN {X 0,Y 731.936,Z 729.943,A -85,B 0,C 180,E1 1697.171,E2 1697.171} C_VEL
LIN {X 0,Y 731.511,Z 760.235,A -85,B 0,C 180,E1 1701.956,E2 1701.956} C_VEL
LIN {X 0,Y 731.249,Z 776.055,A -85,B 0,C 180,E1 1707.028,E2 1707.028} C_VEL
LIN {X 0,Y 731.632,Z 777.587,A -85,B 0,C 180,E1 1711.782,E2 1711.782} C_VEL
LIN {X 0,Y 730.931,Z 766.48,A -85,B 0,C 180,E1 1716.552,E2 1716.552} C_VEL
LIN {X 0,Y 731.279,Z 743.181,A -85,B 0,C 180,E1 1721.059,E2 1721.059} C_VEL
LIN {X 0,Y 731.827,Z 707.146,A -85,B 0,C 180,E1 1725.279,E2 1725.279} C_VEL
LIN {X 0,Y 732.718,Z 657.863,A -85,B 0,C 180,E1 1729.011,E2 1729.011} C_VEL
LIN {X 0,Y 733.669,Z 599.036,A -85,B 0,C 180,E1 1731.795,E2 1731.795} C_VEL
LIN {X 0,Y 734.348,Z 537.102,A -85,B 0,C 180,E1 1733.37,E2 1733.37} C_VEL
LIN {X 0,Y 732.124,Z 477.807,A -85,B 0,C 180,E1 1734.125,E2 1734.125} C_VEL
LIN {X 0,Y 731.46,Z 474.78,A -85,B 0,C 180,E1 1734.283,E2 1734.283} C_VEL
LIN {X 0,Y 730.682,Z 474.78,A -85,B 0,C 180,E1 1740.563,E2 1740.563} C_VEL
LIN {X 0,Y 730.633,Z 474.78,A -85,B 0,C 180,E1 1746.86,E2 1746.86} C_VEL
LIN {X 0,Y 730.466,Z 474.78,A -85,B 0,C 180,E1 1754.176,E2 1754.176} C_VEL
LIN {X 0,Y 730.796,Z 474.78,A -85,B 0,C 180,E1 1762.188,E2 1762.188} C_VEL
LIN {X 0,Y 730.522,Z 474.78,A -85,B 0,C 180,E1 1769.372,E2 1769.372} C_VEL
LIN {X 0,Y 730.246,Z 474.78,A -85,B 0,C 180,E1 1776.061,E2 1776.061} C_VEL
LIN {X 0,Y 731.131,Z 474.78,A -85,B 0,C 180,E1 1782.451,E2 1782.451} C_VEL
LIN {X 0,Y 730.771,Z 474.78,A -85,B 0,C 180,E1 1791.006,E2 1791.006} C_VEL
LIN {X 0,Y 731.091,Z 474.78,A -85,B 0,C 180,E1 1798.181,E2 1798.181} C_VEL
LIN {X 0,Y 731.307,Z 474.78,A -85,B 0,C 180,E1 1805.321,E2 1805.321} C_VEL
LIN {X 0,Y 730.673,Z 474.78,A -85,B 0,C 180,E1 1813.779,E2 1813.779} C_VEL
LIN {X 0,Y 730.811,Z 474.78,A -85,B 0,C 180,E1 1821.265,E2 1821.265} C_VEL
LIN {X 0,Y 731.118,Z 474.78,A -85,B 0,C 180,E1 1829.147,E2 1829.147} C_VEL
LIN {X 0,Y 730.568,Z 474.78,A -85,B 0,C 180,E1 1836.949,E2 1836.949} C_VEL
LIN {X 0,Y 730.479,Z 474.78,A -85,B 0,C 180,E1 1844.256,E2 1844.256} C_VEL
LIN {X 0,Y 730.819,Z 474.78,A -85,B 0,C 180,E1 1852.256,E2 1852.256} C_VEL
LIN {X 0,Y 730.865,Z 474.78,A -85,B 0,C 180,E1 1858.055,E2 1858.055} C_VEL
LIN {X 0,Y 730.769,Z 474.78,A -85,B 0,C 180,E1 1864.823,E2 1864.823} C_VEL
LIN {X 0,Y 731.176,Z 474.78,A -85,B 0,C 180,E1 1872.498,E2 1872.498} C_VEL
LIN {X 0,Y 730.772,Z 474.78,A -85,B 0,C 180,E1 1881.046,E2 1881.046} C_VEL
LIN {X 0,Y 730.997,Z 474.78,A -85,B 0,C 180,E1 1888.217,E2 1888.217} C_VEL
LIN {X 0,Y 731.235,Z 474.78,A -85,B 0,C 180,E1 1895.355,E2 1895.355} C_VEL
LIN {X 0,Y 730.671,Z 474.78,A -85,B 0,C 180,E1 1903.809,E2 1903.809} C_VEL
LIN {X 0,Y 730.781,Z 474.78,A -85,B 0,C 180,E1 1911.294,E2 1911.294} C_VEL
LIN {X 0,Y 730.934,Z 474.78,A -85,B 0,C 180,E1 1919.18,E2 1919.18} C_VEL
LIN {X 0,Y 730.651,Z 474.78,A -85,B 0,C 180,E1 1927.755,E2 1927.755} C_VEL
LIN {X 0,Y 730.805,Z 474.78,A -85,B 0,C 180,E1 1935.983,E2 1935.983} C_VEL
LIN {X 0,Y 730.73,Z 474.78,A -85,B 0,C 180,E1 1943.763,E2 1943.763} C_VEL
LIN {X 0,Y 730.65,Z 474.78,A -85,B 0,C 180,E1 1951.897,E2 1951.897} C_VEL
LIN {X 0,Y 730.983,Z 474.78,A -85,B 0,C 180,E1 1958.74,E2 1958.74} C_VEL
LIN {X 0,Y 731.331,Z 474.78,A -85,B 0,C 180,E1 1967.455,E2 1967.455} C_VEL
LIN {X 0,Y 731.727,Z 474.78,A -85,B 0,C 180,E1 1977.064,E2 1977.064} C_VEL
LIN {X 0,Y 731.261,Z 474.78,A -85,B 0,C 180,E1 1985.393,E2 1985.393} C_VEL
LIN {X 0,Y 730.319,Z 474.78,A -85,B 0,C 180,E1 1987.314,E2 1987.314} C_VEL
LIN {X 0,Y 722.443,Z 474.78,A -85,B 0,C 180,E1 1990.048,E2 1990.048} C_VEL
LIN {X 0,Y 722.147,Z 474.78,A -85,B 0,C 180,E1 1995.263,E2 1995.263} C_VEL
LIN {X 0,Y 722.599,Z 474.78,A -85,B 0,C 180,E1 2001.597,E2 2001.597} C_VEL
LIN {X 0,Y 722.757,Z 474.78,A -85,B 0,C 180,E1 2009.6,E2 2009.6} C_VEL
LIN {X 0,Y 722.453,Z 474.78,A -85,B 0,C 180,E1 2018.327,E2 2018.327} C_VEL
LIN {X 0,Y 722.621,Z 474.78,A -85,B 0,C 180,E1 2026.468,E2 2026.468} C_VEL
LIN {X 0,Y 722.818,Z 474.78,A -85,B 0,C 180,E1 2033.974,E2 2033.974} C_VEL
LIN {X 0,Y 722.599,Z 474.78,A -85,B 0,C 180,E1 2041.823,E2 2041.823} C_VEL
LIN {X 0,Y 723.207,Z 475.65,A -85,B 0,C 180,E1 2045.535,E2 2045.535} C_VEL
LIN {X 0,Y 726.919,Z 503.62,A -85,B 0,C 180,E1 2045.965,E2 2045.965} C_VEL
LIN {X 0,Y 726.485,Z 572.558,A -85,B 0,C 180,E1 2047.135,E2 2047.135} C_VEL
LIN {X 0,Y 725.648,Z 633.315,A -85,B 0,C 180,E1 2049.43,E2 2049.43} C_VEL
LIN {X 0,Y 724.672,Z 687.143,A -85,B 0,C 180,E1 2052.82,E2 2052.82} C_VEL
LIN {X 0,Y 724.066,Z 729.874,A -85,B 0,C 180,E1 2057.019,E2 2057.019} C_VEL
LIN {X 0,Y 723.577,Z 760.238,A -85,B 0,C 180,E1 2061.867,E2 2061.867} C_VEL
LIN {X 0,Y 723.26,Z 776.057,A -85,B 0,C 180,E1 2066.995,E2 2066.995} C_VEL
LIN {X 0,Y 723.628,Z 777.59,A -85,B 0,C 180,E1 2071.801,E2 2071.801} C_VEL
LIN {X 0,Y 722.951,Z 766.484,A -85,B 0,C 180,E1 2076.625,E2 2076.625} C_VEL
LIN {X 0,Y 723.348,Z 743.174,A -85,B 0,C 180,E1 2081.182,E2 2081.182} C_VEL
LIN {X 0,Y 723.97,Z 707.151,A -85,B 0,C 180,E1 2085.449,E2 2085.449} C_VEL
LIN {X 0,Y 725.065,Z 657.379,A -85,B 0,C 180,E1 2089.251,E2 2089.251} C_VEL
LIN {X 0,Y 726.185,Z 597.743,A -85,B 0,C 180,E1 2092.079,E2 2092.079} C_VEL
LIN {X 0,Y 727.024,Z 533.832,A -85,B 0,C 180,E1 2093.674,E2 2093.674} C_VEL
LIN {X 0,Y 724.959,Z 480.044,A -85,B 0,C 180,E1 2094.355,E2 2094.355} C_VEL
LIN {X 0,Y 723.367,Z 474.78,A -85,B 0,C 180,E1 2094.625,E2 2094.625} C_VEL
LIN {X 0,Y 722.583,Z 474.78,A -85,B 0,C 180,E1 2102.355,E2 2102.355} C_VEL
LIN {X 0,Y 722.481,Z 474.78,A -85,B 0,C 180,E1 2109.806,E2 2109.806} C_VEL
LIN {X 0,Y 722.019,Z 474.78,A -85,B 0,C 180,E1 2116.877,E2 2116.877} C_VEL
LIN {X 0,Y 722.611,Z 474.78,A -85,B 0,C 180,E1 2123.2,E2 2123.2} C_VEL
LIN {X 0,Y 722.407,Z 474.78,A -85,B 0,C 180,E1 2130.384,E2 2130.384} C_VEL
LIN {X 0,Y 721.946,Z 474.78,A -85,B 0,C 180,E1 2137.082,E2 2137.082} C_VEL
LIN {X 0,Y 722.604,Z 474.78,A -85,B 0,C 180,E1 2143.496,E2 2143.496} C_VEL
LIN {X 0,Y 722.833,Z 474.78,A -85,B 0,C 180,E1 2150.906,E2 2150.906} C_VEL
LIN {X 0,Y 723.094,Z 474.78,A -85,B 0,C 180,E1 2158.16,E2 2158.16} C_VEL
LIN {X 0,Y 723.257,Z 474.78,A -85,B 0,C 180,E1 2165.381,E2 2165.381} C_VEL
LIN {X 0,Y 722.591,Z 474.78,A -85,B 0,C 180,E1 2173.936,E2 2173.936} C_VEL
LIN {X 0,Y 722.677,Z 474.78,A -85,B 0,C 180,E1 2181.517,E2 2181.517} C_VEL
LIN {X 0,Y 722.97,Z 474.78,A -85,B 0,C 180,E1 2189.508,E2 2189.508} C_VEL
LIN {X 0,Y 722.652,Z 474.78,A -85,B 0,C 180,E1 2196.708,E2 2196.708} C_VEL
LIN {X 0,Y 722.71,Z 474.78,A -85,B 0,C 180,E1 2203.621,E2 2203.621} C_VEL
LIN {X 0,Y 722.949,Z 474.78,A -85,B 0,C 180,E1 2211.847,E2 2211.847} C_VEL
LIN {X 0,Y 722.549,Z 474.78,A -85,B 0,C 180,E1 2219.056,E2 2219.056} C_VEL
LIN {X 0,Y 722.289,Z 474.78,A -85,B 0,C 180,E1 2225.939,E2 2225.939} C_VEL
LIN {X 0,Y 722.59,Z 474.78,A -85,B 0,C 180,E1 2233.541,E2 2233.541} C_VEL
LIN {X 0,Y 722.824,Z 474.78,A -85,B 0,C 180,E1 2240.947,E2 2240.947} C_VEL
LIN {X 0,Y 723,Z 474.78,A -85,B 0,C 180,E1 2248.197,E2 2248.197} C_VEL
LIN {X 0,Y 723.187,Z 474.78,A -85,B 0,C 180,E1 2255.415,E2 2255.415} C_VEL
LIN {X 0,Y 722.586,Z 474.78,A -85,B 0,C 180,E1 2263.966,E2 2263.966} C_VEL
LIN {X 0,Y 722.657,Z 474.78,A -85,B 0,C 180,E1 2271.545,E2 2271.545} C_VEL
LIN {X 0,Y 722.734,Z 474.78,A -85,B 0,C 180,E1 2279.544,E2 2279.544} C_VEL
LIN {X 0,Y 722.415,Z 474.78,A -85,B 0,C 180,E1 2288.262,E2 2288.262} C_VEL
LIN {X 0,Y 722.613,Z 474.78,A -85,B 0,C 180,E1 2296.388,E2 2296.388} C_VEL
LIN {X 0,Y 722.689,Z 474.78,A -85,B 0,C 180,E1 2303.89,E2 2303.89} C_VEL
LIN {X 0,Y 722.682,Z 474.78,A -85,B 0,C 180,E1 2311.853,E2 2311.853} C_VEL
LIN {X 0,Y 722.557,Z 474.78,A -85,B 0,C 180,E1 2319.767,E2 2319.767} C_VEL
LIN {X 0,Y 723.321,Z 474.78,A -85,B 0,C 180,E1 2327.314,E2 2327.314} C_VEL
LIN {X 0,Y 723.686,Z 474.78,A -85,B 0,C 180,E1 2337.032,E2 2337.032} C_VEL
LIN {X 0,Y 723.233,Z 474.78,A -85,B 0,C 180,E1 2345.453,E2 2345.453} C_VEL
LIN {X 0,Y 722.443,Z 474.78,A -85,B 0,C 180,E1 2350.048,E2 2350.048} C_VEL
LIN {X 0,Y 715.17,Z 474.78,A -85,B 0,C 180,E1 2352.827,E2 2352.827} C_VEL
LIN {X 0,Y 714.949,Z 474.78,A -85,B 0,C 180,E1 2360.535,E2 2360.535} C_VEL
LIN {X 0,Y 714.558,Z 474.78,A -85,B 0,C 180,E1 2369.974,E2 2369.974} C_VEL
LIN {X 0,Y 714.73,Z 474.78,A -85,B 0,C 180,E1 2377.282,E2 2377.282} C_VEL
LIN {X 0,Y 714.656,Z 474.78,A -85,B 0,C 180,E1 2386.398,E2 2386.398} C_VEL
LIN {X 0,Y 714.631,Z 474.78,A -85,B 0,C 180,E1 2394.887,E2 2394.887} C_VEL
LIN {X 0,Y 714.606,Z 474.78,A -85,B 0,C 180,E1 2401.853,E2 2401.853} C_VEL
LIN {X 0,Y 715.09,Z 475.449,A -85,B 0,C 180,E1 2405.237,E2 2405.237} C_VEL
LIN {X 0,Y 719.61,Z 502.269,A -85,B 0,C 180,E1 2405.691,E2 2405.691} C_VEL
LIN {X 0,Y 719.128,Z 572.133,A -85,B 0,C 180,E1 2406.876,E2 2406.876} C_VEL
LIN {X 0,Y 718.079,Z 632.673,A -85,B 0,C 180,E1 2409.169,E2 2409.169} C_VEL
LIN {X 0,Y 716.951,Z 686.486,A -85,B 0,C 180,E1 2412.575,E2 2412.575} C_VEL
LIN {X 0,Y 716.179,Z 729.633,A -85,B 0,C 180,E1 2416.842,E2 2416.842} C_VEL
LIN {X 0,Y 715.626,Z 760.242,A -85,B 0,C 180,E1 2421.776,E2 2421.776} C_VEL
LIN {X 0,Y 715.283,Z 776.057,A -85,B 0,C 180,E1 2426.962,E2 2426.962} C_VEL
LIN {X 0,Y 715.624,Z 777.594,A -85,B 0,C 180,E1 2431.821,E2 2431.821} C_VEL
LIN {X 0,Y 714.969,Z 766.488,A -85,B 0,C 180,E1 2436.699,E2 2436.699} C_VEL
LIN {X 0,Y 715.394,Z 743.167,A -85,B 0,C 180,E1 2441.308,E2 2441.308} C_VEL
LIN {X 0,Y 716.099,Z 706.735,A -85,B 0,C 180,E1 2445.665,E2 2445.665} C_VEL
LIN {X 0,Y 717.385,Z 656.331,A -85,B 0,C 180,E1 2449.528,E2 2449.528} C_VEL
LIN {X 0,Y 718.718,Z 597.707,A -85,B 0,C 180,E1 2452.321,E2 2452.321} C_VEL
LIN {X 0,Y 719.684,Z 535.075,A -85,B 0,C 180,E1 2453.91,E2 2453.91} C_VEL
LIN {X 0,Y 717.722,Z 482.221,A -85,B 0,C 180,E1 2454.593,E2 2454.593} C_VEL
LIN {X 0,Y 715.347,Z 474.78,A -85,B 0,C 180,E1 2454.918,E2 2454.918} C_VEL
LIN {X 0,Y 714.68,Z 474.78,A -85,B 0,C 180,E1 2462.945,E2 2462.945} C_VEL
LIN {X 0,Y 714.78,Z 474.78,A -85,B 0,C 180,E1 2471.047,E2 2471.047} C_VEL
LIN {X 0,Y 714.939,Z 474.78,A -85,B 0,C 180,E1 2480.734,E2 2480.734} C_VEL
LIN {X 0,Y 714.667,Z 474.78,A -85,B 0,C 180,E1 2488.617,E2 2488.617} C_VEL
LIN {X 0,Y 714.449,Z 474.78,A -85,B 0,C 180,E1 2495.497,E2 2495.497} C_VEL
LIN {X 0,Y 714.699,Z 474.78,A -85,B 0,C 180,E1 2503.308,E2 2503.308} C_VEL
LIN {X 0,Y 714.855,Z 474.78,A -85,B 0,C 180,E1 2510.804,E2 2510.804} C_VEL
LIN {X 0,Y 715.098,Z 474.78,A -85,B 0,C 180,E1 2518.14,E2 2518.14} C_VEL
LIN {X 0,Y 715.205,Z 474.78,A -85,B 0,C 180,E1 2525.441,E2 2525.441} C_VEL
LIN {X 0,Y 715.174,Z 474.78,A -85,B 0,C 180,E1 2532.833,E2 2532.833} C_VEL
LIN {X 0,Y 714.519,Z 474.78,A -85,B 0,C 180,E1 2541.775,E2 2541.775} C_VEL
LIN {X 0,Y 714.822,Z 474.78,A -85,B 0,C 180,E1 2549.878,E2 2549.878} C_VEL
LIN {X 0,Y 714.483,Z 474.78,A -85,B 0,C 180,E1 2557.256,E2 2557.256} C_VEL
LIN {X 0,Y 714.724,Z 474.78,A -85,B 0,C 180,E1 2563.573,E2 2563.573} C_VEL
LIN {X 0,Y 714.953,Z 474.78,A -85,B 0,C 180,E1 2571.265,E2 2571.265} C_VEL
LIN {X 0,Y 714.667,Z 474.78,A -85,B 0,C 180,E1 2578.676,E2 2578.676} C_VEL
LIN {X 0,Y 714.419,Z 474.78,A -85,B 0,C 180,E1 2585.549,E2 2585.549} C_VEL
LIN {X 0,Y 714.678,Z 474.78,A -85,B 0,C 180,E1 2593.354,E2 2593.354} C_VEL
LIN {X 0,Y 714.847,Z 474.78,A -85,B 0,C 180,E1 2600.845,E2 2600.845} C_VEL
LIN {X 0,Y 715.004,Z 474.78,A -85,B 0,C 180,E1 2608.177,E2 2608.177} C_VEL
LIN {X 0,Y 715.136,Z 474.78,A -85,B 0,C 180,E1 2615.476,E2 2615.476} C_VEL
LIN {X 0,Y 715.202,Z 474.78,A -85,B 0,C 180,E1 2622.864,E2 2622.864} C_VEL
LIN {X 0,Y 714.502,Z 474.78,A -85,B 0,C 180,E1 2631.804,E2 2631.804} C_VEL
LIN {X 0,Y 714.524,Z 474.78,A -85,B 0,C 180,E1 2639.918,E2 2639.918} C_VEL
LIN {X 0,Y 714.632,Z 474.78,A -85,B 0,C 180,E1 2647.296,E2 2647.296} C_VEL
LIN {X 0,Y 714.596,Z 474.78,A -85,B 0,C 180,E1 2656.418,E2 2656.418} C_VEL
LIN {X 0,Y 714.362,Z 474.78,A -85,B 0,C 180,E1 2664.815,E2 2664.815} C_VEL
LIN {X 0,Y 714.698,Z 474.78,A -85,B 0,C 180,E1 2671.711,E2 2671.711} C_VEL
LIN {X 0,Y 714.644,Z 474.78,A -85,B 0,C 180,E1 2679.533,E2 2679.533} C_VEL
LIN {X 0,Y 715.346,Z 474.78,A -85,B 0,C 180,E1 2687.17,E2 2687.17} C_VEL
LIN {X 0,Y 715.645,Z 474.78,A -85,B 0,C 180,E1 2696.998,E2 2696.998} C_VEL
LIN {X 0,Y 715.182,Z 474.78,A -85,B 0,C 180,E1 2705.515,E2 2705.515} C_VEL
LIN {X 0,Y 715.17,Z 474.78,A -85,B 0,C 180,E1 2712.827,E2 2712.827} C_VEL
LIN {X 0,Y 706.112,Z 474.78,A -85,B 0,C 180,E1 2715.593,E2 2715.593} C_VEL
LIN {X 0,Y 706.326,Z 474.78,A -85,B 0,C 180,E1 2722.12,E2 2722.12} C_VEL
LIN {X 0,Y 706.621,Z 474.78,A -85,B 0,C 180,E1 2729.637,E2 2729.637} C_VEL
LIN {X 0,Y 706.317,Z 474.78,A -85,B 0,C 180,E1 2738.402,E2 2738.402} C_VEL
LIN {X 0,Y 706.745,Z 474.78,A -85,B 0,C 180,E1 2746.039,E2 2746.039} C_VEL
LIN {X 0,Y 706.764,Z 474.78,A -85,B 0,C 180,E1 2753.839,E2 2753.839} C_VEL
LIN {X 0,Y 706.708,Z 474.78,A -85,B 0,C 180,E1 2761.131,E2 2761.131} C_VEL
LIN {X 0,Y 707.069,Z 476.019,A -85,B 0,C 180,E1 2764.943,E2 2764.943} C_VEL
LIN {X 0,Y 712.327,Z 502.667,A -85,B 0,C 180,E1 2765.43,E2 2765.43} C_VEL
LIN {X 0,Y 711.742,Z 572.119,A -85,B 0,C 180,E1 2766.622,E2 2766.622} C_VEL
LIN {X 0,Y 710.494,Z 633.224,A -85,B 0,C 180,E1 2768.966,E2 2768.966} C_VEL
LIN {X 0,Y 709.174,Z 686.947,A -85,B 0,C 180,E1 2772.416,E2 2772.416} C_VEL
LIN {X 0,Y 708.288,Z 729.637,A -85,B 0,C 180,E1 2776.693,E2 2776.693} C_VEL
LIN {X 0,Y 707.697,Z 760.246,A -85,B 0,C 180,E1 2781.683,E2 2781.683} C_VEL
LIN {X 0,Y 707.295,Z 776.055,A -85,B 0,C 180,E1 2786.927,E2 2786.927} C_VEL
LIN {X 0,Y 707.621,Z 777.596,A -85,B 0,C 180,E1 2791.842,E2 2791.842} C_VEL
LIN {X 0,Y 706.993,Z 766.492,A -85,B 0,C 180,E1 2796.775,E2 2796.775} C_VEL
LIN {X 0,Y 707.472,Z 743.16,A -85,B 0,C 180,E1 2801.436,E2 2801.436} C_VEL
LIN {X 0,Y 708.279,Z 706.74,A -85,B 0,C 180,E1 2805.842,E2 2805.842} C_VEL
LIN {X 0,Y 709.705,Z 657.982,A -85,B 0,C 180,E1 2809.646,E2 2809.646} C_VEL
LIN {X 0,Y 711.252,Z 598.855,A -85,B 0,C 180,E1 2812.527,E2 2812.527} C_VEL
LIN {X 0,Y 712.385,Z 535.563,A -85,B 0,C 180,E1 2814.163,E2 2814.163} C_VEL
LIN {X 0,Y 710.301,Z 483.921,A -85,B 0,C 180,E1 2814.849,E2 2814.849} C_VEL
LIN {X 0,Y 707.316,Z 474.78,A -85,B 0,C 180,E1 2815.147,E2 2815.147} C_VEL
LIN {X 0,Y 706.721,Z 474.78,A -85,B 0,C 180,E1 2823.174,E2 2823.174} C_VEL
LIN {X 0,Y 706.928,Z 474.78,A -85,B 0,C 180,E1 2832.176,E2 2832.176} C_VEL
LIN {X 0,Y 706.806,Z 474.78,A -85,B 0,C 180,E1 2841.548,E2 2841.548} C_VEL
LIN {X 0,Y 706.713,Z 474.78,A -85,B 0,C 180,E1 2848.222,E2 2848.222} C_VEL
LIN {X 0,Y 706.292,Z 474.78,A -85,B 0,C 180,E1 2855.856,E2 2855.856} C_VEL
LIN {X 0,Y 706.734,Z 474.78,A -85,B 0,C 180,E1 2863.114,E2 2863.114} C_VEL
LIN {X 0,Y 706.891,Z 474.78,A -85,B 0,C 180,E1 2870.699,E2 2870.699} C_VEL
LIN {X 0,Y 707.102,Z 474.78,A -85,B 0,C 180,E1 2878.119,E2 2878.119} C_VEL
LIN {X 0,Y 707.173,Z 474.78,A -85,B 0,C 180,E1 2885.503,E2 2885.503} C_VEL
LIN {X 0,Y 707.086,Z 474.78,A -85,B 0,C 180,E1 2892.983,E2 2892.983} C_VEL
LIN {X 0,Y 706.742,Z 474.78,A -85,B 0,C 180,E1 2901.029,E2 2901.029} C_VEL
LIN {X 0,Y 706.74,Z 474.78,A -85,B 0,C 180,E1 2910.255,E2 2910.255} C_VEL
LIN {X 0,Y 706.406,Z 474.78,A -85,B 0,C 180,E1 2917.696,E2 2917.696} C_VEL
LIN {X 0,Y 706.469,Z 474.78,A -85,B 0,C 180,E1 2924.213,E2 2924.213} C_VEL
LIN {X 0,Y 706.755,Z 474.78,A -85,B 0,C 180,E1 2932.3,E2 2932.3} C_VEL
LIN {X 0,Y 706.444,Z 474.78,A -85,B 0,C 180,E1 2939.704,E2 2939.704} C_VEL
LIN {X 0,Y 706.072,Z 474.78,A -85,B 0,C 180,E1 2946.588,E2 2946.588} C_VEL
LIN {X 0,Y 706.723,Z 474.78,A -85,B 0,C 180,E1 2953.161,E2 2953.161} C_VEL
LIN {X 0,Y 706.883,Z 474.78,A -85,B 0,C 180,E1 2960.741,E2 2960.741} C_VEL
LIN {X 0,Y 707.008,Z 474.78,A -85,B 0,C 180,E1 2968.156,E2 2968.156} C_VEL
LIN {X 0,Y 707.104,Z 474.78,A -85,B 0,C 180,E1 2975.538,E2 2975.538} C_VEL
LIN {X 0,Y 707.096,Z 474.78,A -85,B 0,C 180,E1 2983.014,E2 2983.014} C_VEL
LIN {X 0,Y 706.732,Z 474.78,A -85,B 0,C 180,E1 2991.058,E2 2991.058} C_VEL
LIN {X 0,Y 706.568,Z 474.78,A -85,B 0,C 180,E1 2999.656,E2 2999.656} C_VEL
LIN {X 0,Y 706.272,Z 474.78,A -85,B 0,C 180,E1 3008.423,E2 3008.423} C_VEL
LIN {X 0,Y 706.703,Z 474.78,A -85,B 0,C 180,E1 3015.961,E2 3015.961} C_VEL
LIN {X 0,Y 706.551,Z 474.78,A -85,B 0,C 180,E1 3023.852,E2 3023.852} C_VEL
LIN {X 0,Y 706.725,Z 474.78,A -85,B 0,C 180,E1 3031.158,E2 3031.158} C_VEL
LIN {X 0,Y 706.677,Z 474.78,A -85,B 0,C 180,E1 3039.292,E2 3039.292} C_VEL
LIN {X 0,Y 707.34,Z 474.78,A -85,B 0,C 180,E1 3047.288,E2 3047.288} C_VEL
LIN {X 0,Y 707.605,Z 474.78,A -85,B 0,C 180,E1 3056.964,E2 3056.964} C_VEL
LIN {X 0,Y 707.146,Z 474.78,A -85,B 0,C 180,E1 3065.578,E2 3065.578} C_VEL
LIN {X 0,Y 707.076,Z 474.78,A -85,B 0,C 180,E1 3073.059,E2 3073.059} C_VEL
LIN {X 0,Y 706.112,Z 474.78,A -85,B 0,C 180,E1 3075.593,E2 3075.593} C_VEL
LIN {X 0,Y 698.46,Z 474.78,A -85,B 0,C 180,E1 3078.418,E2 3078.418} C_VEL
LIN {X 0,Y 698.339,Z 474.78,A -85,B 0,C 180,E1 3086.49,E2 3086.49} C_VEL
LIN {X 0,Y 698.123,Z 474.78,A -85,B 0,C 180,E1 3093.699,E2 3093.699} C_VEL
LIN {X 0,Y 697.974,Z 474.78,A -85,B 0,C 180,E1 3099.934,E2 3099.934} C_VEL
LIN {X 0,Y 698.441,Z 474.78,A -85,B 0,C 180,E1 3106.847,E2 3106.847} C_VEL
LIN {X 0,Y 698.56,Z 474.78,A -85,B 0,C 180,E1 3114.881,E2 3114.881} C_VEL
LIN {X 0,Y 698.527,Z 474.78,A -85,B 0,C 180,E1 3122.176,E2 3122.176} C_VEL
LIN {X 0,Y 698.976,Z 475.919,A -85,B 0,C 180,E1 3124.631,E2 3124.631} C_VEL
LIN {X 0,Y 705.043,Z 498.781,A -85,B 0,C 180,E1 3125.116,E2 3125.116} C_VEL
LIN {X 0,Y 704.479,Z 569.632,A -85,B 0,C 180,E1 3126.292,E2 3126.292} C_VEL
LIN {X 0,Y 702.971,Z 630.989,A -85,B 0,C 180,E1 3128.615,E2 3128.615} C_VEL
LIN {X 0,Y 701.494,Z 685.316,A -85,B 0,C 180,E1 3132.084,E2 3132.084} C_VEL
LIN {X 0,Y 700.38,Z 728.375,A -85,B 0,C 180,E1 3136.381,E2 3136.381} C_VEL
LIN {X 0,Y 699.843,Z 759.116,A -85,B 0,C 180,E1 3141.343,E2 3141.343} C_VEL
LIN {X 0,Y 699.507,Z 775.119,A -85,B 0,C 180,E1 3146.369,E2 3146.369} C_VEL
LIN {X 0,Y 699.646,Z 777.594,A -85,B 0,C 180,E1 3151.863,E2 3151.863} C_VEL
LIN {X 0,Y 699.019,Z 766.496,A -85,B 0,C 180,E1 3156.853,E2 3156.853} C_VEL
LIN {X 0,Y 699.562,Z 743.154,A -85,B 0,C 180,E1 3161.567,E2 3161.567} C_VEL
LIN {X 0,Y 700.433,Z 706.741,A -85,B 0,C 180,E1 3166.024,E2 3166.024} C_VEL
LIN {X 0,Y 702.061,Z 657.495,A -85,B 0,C 180,E1 3169.899,E2 3169.899} C_VEL
LIN {X 0,Y 703.801,Z 598.848,A -85,B 0,C 180,E1 3172.779,E2 3172.779} C_VEL
LIN {X 0,Y 705.082,Z 536.224,A -85,B 0,C 180,E1 3174.418,E2 3174.418} C_VEL
LIN {X 0,Y 703.119,Z 486.011,A -85,B 0,C 180,E1 3175.097,E2 3175.097} C_VEL
LIN {X 0,Y 699.293,Z 474.78,A -85,B 0,C 180,E1 3175.532,E2 3175.532} C_VEL
LIN {X 0,Y 698.809,Z 474.78,A -85,B 0,C 180,E1 3183.599,E2 3183.599} C_VEL
LIN {X 0,Y 698.769,Z 474.78,A -85,B 0,C 180,E1 3191.446,E2 3191.446} C_VEL
LIN {X 0,Y 698.906,Z 474.78,A -85,B 0,C 180,E1 3200.379,E2 3200.379} C_VEL
LIN {X 0,Y 698.809,Z 474.78,A -85,B 0,C 180,E1 3207.82,E2 3207.82} C_VEL
LIN {X 0,Y 698.586,Z 474.78,A -85,B 0,C 180,E1 3214.903,E2 3214.903} C_VEL
LIN {X 0,Y 698.803,Z 474.78,A -85,B 0,C 180,E1 3222.917,E2 3222.917} C_VEL
LIN {X 0,Y 698.815,Z 474.78,A -85,B 0,C 180,E1 3230.89,E2 3230.89} C_VEL
LIN {X 0,Y 699.125,Z 474.78,A -85,B 0,C 180,E1 3238.097,E2 3238.097} C_VEL
LIN {X 0,Y 699.121,Z 474.78,A -85,B 0,C 180,E1 3245.567,E2 3245.567} C_VEL
LIN {X 0,Y 698.984,Z 474.78,A -85,B 0,C 180,E1 3253.136,E2 3253.136} C_VEL
LIN {X 0,Y 698.79,Z 474.78,A -85,B 0,C 180,E1 3260.953,E2 3260.953} C_VEL
LIN {X 0,Y 698.885,Z 474.78,A -85,B 0,C 180,E1 3269.196,E2 3269.196} C_VEL
LIN {X 0,Y 698.649,Z 474.78,A -85,B 0,C 180,E1 3276.623,E2 3276.623} C_VEL
LIN {X 0,Y 698.676,Z 474.78,A -85,B 0,C 180,E1 3283.354,E2 3283.354} C_VEL
LIN {X 0,Y 698.756,Z 474.78,A -85,B 0,C 180,E1 3292.361,E2 3292.361} C_VEL
LIN {X 0,Y 698.475,Z 474.78,A -85,B 0,C 180,E1 3299.322,E2 3299.322} C_VEL
LIN {X 0,Y 698.168,Z 474.78,A -85,B 0,C 180,E1 3306.307,E2 3306.307} C_VEL
LIN {X 0,Y 698.794,Z 474.78,A -85,B 0,C 180,E1 3312.964,E2 3312.964} C_VEL
LIN {X 0,Y 698.842,Z 474.78,A -85,B 0,C 180,E1 3320.813,E2 3320.813} C_VEL
LIN {X 0,Y 699.029,Z 474.78,A -85,B 0,C 180,E1 3328.135,E2 3328.135} C_VEL
LIN {X 0,Y 699.054,Z 474.78,A -85,B 0,C 180,E1 3335.602,E2 3335.602} C_VEL
LIN {X 0,Y 698.991,Z 474.78,A -85,B 0,C 180,E1 3343.168,E2 3343.168} C_VEL
LIN {X 0,Y 698.78,Z 474.78,A -85,B 0,C 180,E1 3350.982,E2 3350.982} C_VEL
LIN {X 0,Y 698.668,Z 474.78,A -85,B 0,C 180,E1 3359.234,E2 3359.234} C_VEL
LIN {X 0,Y 698.312,Z 474.78,A -85,B 0,C 180,E1 3368.237,E2 3368.237} C_VEL
LIN {X 0,Y 698.376,Z 474.78,A -85,B 0,C 180,E1 3376.868,E2 3376.868} C_VEL
LIN {X 0,Y 698.276,Z 474.78,A -85,B 0,C 180,E1 3384.89,E2 3384.89} C_VEL
LIN {X 0,Y 698.475,Z 474.78,A -85,B 0,C 180,E1 3392.201,E2 3392.201} C_VEL
LIN {X 0,Y 698.755,Z 474.78,A -85,B 0,C 180,E1 3399.046,E2 3399.046} C_VEL
LIN {X 0,Y 699.404,Z 474.78,A -85,B 0,C 180,E1 3408.145,E2 3408.145} C_VEL
LIN {X 0,Y 699.101,Z 474.78,A -85,B 0,C 180,E1 3418.172,E2 3418.172} C_VEL
LIN {X 0,Y 699.095,Z 474.78,A -85,B 0,C 180,E1 3425.642,E2 3425.642} C_VEL
LIN {X 0,Y 698.973,Z 474.78,A -85,B 0,C 180,E1 3433.213,E2 3433.213} C_VEL
LIN {X 0,Y 698.46,Z 474.78,A -85,B 0,C 180,E1 3438.418,E2 3438.418} C_VEL
LIN {X 0,Y 690.612,Z 474.78,A -85,B 0,C 180,E1 3441.282,E2 3441.282} C_VEL
LIN {X 0,Y 690.499,Z 474.78,A -85,B 0,C 180,E1 3449.83,E2 3449.83} C_VEL
LIN {X 0,Y 690.568,Z 474.78,A -85,B 0,C 180,E1 3457.218,E2 3457.218} C_VEL
LIN {X 0,Y 690.517,Z 474.78,A -85,B 0,C 180,E1 3466.228,E2 3466.228} C_VEL
LIN {X 0,Y 690.63,Z 474.78,A -85,B 0,C 180,E1 3474.416,E2 3474.416} C_VEL
LIN {X 0,Y 690.601,Z 474.78,A -85,B 0,C 180,E1 3481.828,E2 3481.828} C_VEL
LIN {X 0,Y 690.917,Z 476.334,A -85,B 0,C 180,E1 3484.318,E2 3484.318} C_VEL
LIN {X 0,Y 697.797,Z 498.804,A -85,B 0,C 180,E1 3484.84,E2 3484.84} C_VEL
LIN {X 0,Y 697.151,Z 569.392,A -85,B 0,C 180,E1 3486.021,E2 3486.021} C_VEL
LIN {X 0,Y 695.47,Z 630.348,A -85,B 0,C 180,E1 3488.34,E2 3488.34} C_VEL
LIN {X 0,Y 693.772,Z 683.466,A -85,B 0,C 180,E1 3491.732,E2 3491.732} C_VEL
LIN {X 0,Y 692.435,Z 727.049,A -85,B 0,C 180,E1 3496.06,E2 3496.06} C_VEL
LIN {X 0,Y 691.894,Z 758.254,A -85,B 0,C 180,E1 3501.061,E2 3501.061} C_VEL
LIN {X 0,Y 691.555,Z 774.934,A -85,B 0,C 180,E1 3506.228,E2 3506.228} C_VEL
LIN {X 0,Y 691.643,Z 777.588,A -85,B 0,C 180,E1 3511.885,E2 3511.885} C_VEL
LIN {X 0,Y 691.068,Z 766.5,A -85,B 0,C 180,E1 3516.932,E2 3516.932} C_VEL
LIN {X 0,Y 691.617,Z 743.147,A -85,B 0,C 180,E1 3521.702,E2 3521.702} C_VEL
LIN {X 0,Y 692.614,Z 706.733,A -85,B 0,C 180,E1 3526.21,E2 3526.21} C_VEL
LIN {X 0,Y 694.498,Z 657.1,A -85,B 0,C 180,E1 3530.149,E2 3530.149} C_VEL
LIN {X 0,Y 696.372,Z 599.018,A -85,B 0,C 180,E1 3533.029,E2 3533.029} C_VEL
LIN {X 0,Y 697.813,Z 536.618,A -85,B 0,C 180,E1 3534.683,E2 3534.683} C_VEL
LIN {X 0,Y 696.046,Z 488.582,A -85,B 0,C 180,E1 3535.342,E2 3535.342} C_VEL
LIN {X 0,Y 691.277,Z 474.78,A -85,B 0,C 180,E1 3535.846,E2 3535.846} C_VEL
LIN {X 0,Y 690.794,Z 474.78,A -85,B 0,C 180,E1 3544.484,E2 3544.484} C_VEL
LIN {X 0,Y 690.64,Z 474.78,A -85,B 0,C 180,E1 3552.558,E2 3552.558} C_VEL
LIN {X 0,Y 690.79,Z 474.78,A -85,B 0,C 180,E1 3561.199,E2 3561.199} C_VEL
LIN {X 0,Y 690.555,Z 474.78,A -85,B 0,C 180,E1 3568.87,E2 3568.87} C_VEL
LIN {X 0,Y 690.222,Z 474.78,A -85,B 0,C 180,E1 3575.964,E2 3575.964} C_VEL
LIN {X 0,Y 690.828,Z 474.78,A -85,B 0,C 180,E1 3582.727,E2 3582.727} C_VEL
LIN {X 0,Y 690.929,Z 474.78,A -85,B 0,C 180,E1 3590.482,E2 3590.482} C_VEL
LIN {X 0,Y 691.129,Z 474.78,A -85,B 0,C 180,E1 3598.075,E2 3598.075} C_VEL
LIN {X 0,Y 691.089,Z 474.78,A -85,B 0,C 180,E1 3605.632,E2 3605.632} C_VEL
LIN {X 0,Y 690.885,Z 474.78,A -85,B 0,C 180,E1 3613.293,E2 3613.293} C_VEL
LIN {X 0,Y 690.658,Z 474.78,A -85,B 0,C 180,E1 3621.211,E2 3621.211} C_VEL
LIN {X 0,Y 690.728,Z 474.78,A -85,B 0,C 180,E1 3629.863,E2 3629.863} C_VEL
LIN {X 0,Y 690.533,Z 474.78,A -85,B 0,C 180,E1 3637.125,E2 3637.125} C_VEL
LIN {X 0,Y 690.353,Z 474.78,A -85,B 0,C 180,E1 3644.445,E2 3644.445} C_VEL
LIN {X 0,Y 690.71,Z 474.78,A -85,B 0,C 180,E1 3652.859,E2 3652.859} C_VEL
LIN {X 0,Y 690.403,Z 474.78,A -85,B 0,C 180,E1 3660.382,E2 3660.382} C_VEL
LIN {X 0,Y 689.971,Z 474.78,A -85,B 0,C 180,E1 3667.379,E2 3667.379} C_VEL
LIN {X 0,Y 690.395,Z 474.78,A -85,B 0,C 180,E1 3674.064,E2 3674.064} C_VEL
LIN {X 0,Y 690.923,Z 474.78,A -85,B 0,C 180,E1 3680.525,E2 3680.525} C_VEL
LIN {X 0,Y 691.033,Z 474.78,A -85,B 0,C 180,E1 3688.114,E2 3688.114} C_VEL
LIN {X 0,Y 691.021,Z 474.78,A -85,B 0,C 180,E1 3695.668,E2 3695.668} C_VEL
LIN {X 0,Y 690.919,Z 474.78,A -85,B 0,C 180,E1 3703.324,E2 3703.324} C_VEL
LIN {X 0,Y 690.647,Z 474.78,A -85,B 0,C 180,E1 3711.241,E2 3711.241} C_VEL
LIN {X 0,Y 690.437,Z 474.78,A -85,B 0,C 180,E1 3719.849,E2 3719.849} C_VEL
LIN {X 0,Y 690.493,Z 474.78,A -85,B 0,C 180,E1 3727.155,E2 3727.155} C_VEL
LIN {X 0,Y 690.485,Z 474.78,A -85,B 0,C 180,E1 3736.251,E2 3736.251} C_VEL
LIN {X 0,Y 690.376,Z 474.78,A -85,B 0,C 180,E1 3744.428,E2 3744.428} C_VEL
LIN {X 0,Y 690.557,Z 474.78,A -85,B 0,C 180,E1 3751.854,E2 3751.854} C_VEL
LIN {X 0,Y 690.426,Z 474.78,A -85,B 0,C 180,E1 3760.126,E2 3760.126} C_VEL
LIN {X 0,Y 691.378,Z 474.78,A -85,B 0,C 180,E1 3768.005,E2 3768.005} C_VEL
LIN {X 0,Y 691.105,Z 474.78,A -85,B 0,C 180,E1 3778.151,E2 3778.151} C_VEL
LIN {X 0,Y 691.076,Z 474.78,A -85,B 0,C 180,E1 3785.708,E2 3785.708} C_VEL
LIN {X 0,Y 690.894,Z 474.78,A -85,B 0,C 180,E1 3793.37,E2 3793.37} C_VEL
LIN {X 0,Y 690.612,Z 474.78,A -85,B 0,C 180,E1 3801.282,E2 3801.282} C_VEL
LIN {X 0,Y 681.889,Z 474.78,A -85,B 0,C 180,E1 3804.156,E2 3804.156} C_VEL
LIN {X 0,Y 682.159,Z 474.78,A -85,B 0,C 180,E1 3811.143,E2 3811.143} C_VEL
LIN {X 0,Y 682.344,Z 474.78,A -85,B 0,C 180,E1 3817.91,E2 3817.91} C_VEL
LIN {X 0,Y 682.487,Z 474.78,A -85,B 0,C 180,E1 3826.316,E2 3826.316} C_VEL
LIN {X 0,Y 682.659,Z 474.78,A -85,B 0,C 180,E1 3834.28,E2 3834.28} C_VEL
LIN {X 0,Y 682.608,Z 474.78,A -85,B 0,C 180,E1 3841.477,E2 3841.477} C_VEL
LIN {X 0,Y 682.766,Z 475.969,A -85,B 0,C 180,E1 3843.985,E2 3843.985} C_VEL
LIN {X 0,Y 690.569,Z 499.97,A -85,B 0,C 180,E1 3844.571,E2 3844.571} C_VEL
LIN {X 0,Y 689.816,Z 569.663,A -85,B 0,C 180,E1 3845.758,E2 3845.758} C_VEL
LIN {X 0,Y 687.92,Z 631.191,A -85,B 0,C 180,E1 3848.133,E2 3848.133} C_VEL
LIN {X 0,Y 686,Z 685.265,A -85,B 0,C 180,E1 3851.661,E2 3851.661} C_VEL
LIN {X 0,Y 684.519,Z 728.364,A -85,B 0,C 180,E1 3856.059,E2 3856.059} C_VEL
LIN {X 0,Y 683.917,Z 758.749,A -85,B 0,C 180,E1 3861.063,E2 3861.063} C_VEL
LIN {X 0,Y 683.559,Z 774.934,A -85,B 0,C 180,E1 3866.184,E2 3866.184} C_VEL
LIN {X 0,Y 683.653,Z 777.582,A -85,B 0,C 180,E1 3871.907,E2 3871.907} C_VEL
LIN {X 0,Y 683.086,Z 766.504,A -85,B 0,C 180,E1 3877.013,E2 3877.013} C_VEL
LIN {X 0,Y 683.731,Z 742.122,A -85,B 0,C 180,E1 3882.001,E2 3882.001} C_VEL
LIN {X 0,Y 684.942,Z 703.369,A -85,B 0,C 180,E1 3886.728,E2 3886.728} C_VEL
LIN {X 0,Y 687.059,Z 652.261,A -85,B 0,C 180,E1 3890.68,E2 3890.68} C_VEL
LIN {X 0,Y 689.072,Z 593.316,A -85,B 0,C 180,E1 3893.495,E2 3893.495} C_VEL
LIN {X 0,Y 690.581,Z 530.159,A -85,B 0,C 180,E1 3895.058,E2 3895.058} C_VEL
LIN {X 0,Y 688.775,Z 490.421,A -85,B 0,C 180,E1 3895.608,E2 3895.608} C_VEL
LIN {X 0,Y 683.269,Z 474.78,A -85,B 0,C 180,E1 3896.11,E2 3896.11} C_VEL
LIN {X 0,Y 682.824,Z 474.78,A -85,B 0,C 180,E1 3904.495,E2 3904.495} C_VEL
LIN {X 0,Y 682.455,Z 474.78,A -85,B 0,C 180,E1 3913.681,E2 3913.681} C_VEL
LIN {X 0,Y 682.62,Z 474.78,A -85,B 0,C 180,E1 3922.274,E2 3922.274} C_VEL
LIN {X 0,Y 682.414,Z 474.78,A -85,B 0,C 180,E1 3929.94,E2 3929.94} C_VEL
LIN {X 0,Y 681.982,Z 474.78,A -85,B 0,C 180,E1 3937.341,E2 3937.341} C_VEL
LIN {X 0,Y 682.423,Z 474.78,A -85,B 0,C 180,E1 3943.825,E2 3943.825} C_VEL
LIN {X 0,Y 682.523,Z 474.78,A -85,B 0,C 180,E1 3951.654,E2 3951.654} C_VEL
LIN {X 0,Y 683.136,Z 474.78,A -85,B 0,C 180,E1 3958.053,E2 3958.053} C_VEL
LIN {X 0,Y 683.038,Z 474.78,A -85,B 0,C 180,E1 3965.698,E2 3965.698} C_VEL
LIN {X 0,Y 682.795,Z 474.78,A -85,B 0,C 180,E1 3973.453,E2 3973.453} C_VEL
LIN {X 0,Y 682.531,Z 474.78,A -85,B 0,C 180,E1 3981.476,E2 3981.476} C_VEL
LIN {X 0,Y 682.725,Z 474.78,A -85,B 0,C 180,E1 3989.957,E2 3989.957} C_VEL
LIN {X 0,Y 682.41,Z 474.78,A -85,B 0,C 180,E1 3997.917,E2 3997.917} C_VEL
LIN {X 0,Y 682.154,Z 474.78,A -85,B 0,C 180,E1 4005.551,E2 4005.551} C_VEL
LIN {X 0,Y 682.691,Z 474.78,A -85,B 0,C 180,E1 4012.348,E2 4012.348} C_VEL
LIN {X 0,Y 682.423,Z 474.78,A -85,B 0,C 180,E1 4020,E2 4020} C_VEL
LIN {X 0,Y 681.976,Z 474.78,A -85,B 0,C 180,E1 4027.309,E2 4027.309} C_VEL
LIN {X 0,Y 682.433,Z 474.78,A -85,B 0,C 180,E1 4033.873,E2 4033.873} C_VEL
LIN {X 0,Y 682.486,Z 474.78,A -85,B 0,C 180,E1 4041.696,E2 4041.696} C_VEL
LIN {X 0,Y 683.04,Z 474.78,A -85,B 0,C 180,E1 4048.092,E2 4048.092} C_VEL
LIN {X 0,Y 682.972,Z 474.78,A -85,B 0,C 180,E1 4055.735,E2 4055.735} C_VEL
LIN {X 0,Y 682.823,Z 474.78,A -85,B 0,C 180,E1 4063.485,E2 4063.485} C_VEL
LIN {X 0,Y 682.521,Z 474.78,A -85,B 0,C 180,E1 4071.507,E2 4071.507} C_VEL
LIN {X 0,Y 682.405,Z 474.78,A -85,B 0,C 180,E1 4080.001,E2 4080.001} C_VEL
LIN {X 0,Y 682.255,Z 474.78,A -85,B 0,C 180,E1 4087.927,E2 4087.927} C_VEL
LIN {X 0,Y 682.487,Z 474.78,A -85,B 0,C 180,E1 4096.232,E2 4096.232} C_VEL
LIN {X 0,Y 682.425,Z 474.78,A -85,B 0,C 180,E1 4104.204,E2 4104.204} C_VEL
LIN {X 0,Y 682.549,Z 474.78,A -85,B 0,C 180,E1 4111.494,E2 4111.494} C_VEL
LIN {X 0,Y 682.467,Z 474.78,A -85,B 0,C 180,E1 4119.884,E2 4119.884} C_VEL
LIN {X 0,Y 683.386,Z 474.78,A -85,B 0,C 180,E1 4127.863,E2 4127.863} C_VEL
LIN {X 0,Y 683.113,Z 474.78,A -85,B 0,C 180,E1 4138.129,E2 4138.129} C_VEL
LIN {X 0,Y 683.025,Z 474.78,A -85,B 0,C 180,E1 4145.775,E2 4145.775} C_VEL
LIN {X 0,Y 682.802,Z 474.78,A -85,B 0,C 180,E1 4153.531,E2 4153.531} C_VEL
LIN {X 0,Y 682.483,Z 474.78,A -85,B 0,C 180,E1 4161.56,E2 4161.56} C_VEL
LIN {X 0,Y 681.889,Z 474.78,A -85,B 0,C 180,E1 4164.156,E2 4164.156} C_VEL
LIN {X 0,Y 674.427,Z 474.78,A -85,B 0,C 180,E1 4167.096,E2 4167.096} C_VEL
LIN {X 0,Y 674.352,Z 474.78,A -85,B 0,C 180,E1 4175.057,E2 4175.057} C_VEL
LIN {X 0,Y 674.405,Z 474.78,A -85,B 0,C 180,E1 4183.38,E2 4183.38} C_VEL
LIN {X 0,Y 674.532,Z 474.78,A -85,B 0,C 180,E1 4191.811,E2 4191.811} C_VEL
LIN {X 0,Y 674.808,Z 474.78,A -85,B 0,C 180,E1 4200.031,E2 4200.031} C_VEL
LIN {X 0,Y 674.758,Z 476.176,A -85,B 0,C 180,E1 4203.657,E2 4203.657} C_VEL
LIN {X 0,Y 683.361,Z 503.244,A -85,B 0,C 180,E1 4204.321,E2 4204.321} C_VEL
LIN {X 0,Y 682.415,Z 572.008,A -85,B 0,C 180,E1 4205.551,E2 4205.551} C_VEL
LIN {X 0,Y 680.354,Z 632.845,A -85,B 0,C 180,E1 4207.967,E2 4207.967} C_VEL
LIN {X 0,Y 678.246,Z 686.46,A -85,B 0,C 180,E1 4211.543,E2 4211.543} C_VEL
LIN {X 0,Y 676.625,Z 729.652,A -85,B 0,C 180,E1 4216.058,E2 4216.058} C_VEL
LIN {X 0,Y 675.889,Z 760.244,A -85,B 0,C 180,E1 4221.285,E2 4221.285} C_VEL
LIN {X 0,Y 675.403,Z 776.035,A -85,B 0,C 180,E1 4226.782,E2 4226.782} C_VEL
LIN {X 0,Y 675.655,Z 777.576,A -85,B 0,C 180,E1 4231.929,E2 4231.929} C_VEL
LIN {X 0,Y 675.107,Z 766.508,A -85,B 0,C 180,E1 4237.097,E2 4237.097} C_VEL
LIN {X 0,Y 675.758,Z 743.372,A -85,B 0,C 180,E1 4241.942,E2 4241.942} C_VEL
LIN {X 0,Y 676.998,Z 706.715,A -85,B 0,C 180,E1 4246.595,E2 4246.595} C_VEL
LIN {X 0,Y 679.258,Z 657.621,A -85,B 0,C 180,E1 4250.587,E2 4250.587} C_VEL
LIN {X 0,Y 681.543,Z 598.855,A -85,B 0,C 180,E1 4253.565,E2 4253.565} C_VEL
LIN {X 0,Y 683.274,Z 536.817,A -85,B 0,C 180,E1 4255.241,E2 4255.241} C_VEL
LIN {X 0,Y 681.702,Z 492.736,A -85,B 0,C 180,E1 4255.866,E2 4255.866} C_VEL
LIN {X 0,Y 675.254,Z 474.78,A -85,B 0,C 180,E1 4256.511,E2 4256.511} C_VEL
LIN {X 0,Y 674.779,Z 474.78,A -85,B 0,C 180,E1 4264.965,E2 4264.965} C_VEL
LIN {X 0,Y 674.512,Z 474.78,A -85,B 0,C 180,E1 4273.292,E2 4273.292} C_VEL
LIN {X 0,Y 674.64,Z 474.78,A -85,B 0,C 180,E1 4281.748,E2 4281.748} C_VEL
LIN {X 0,Y 674.448,Z 474.78,A -85,B 0,C 180,E1 4289.547,E2 4289.547} C_VEL
LIN {X 0,Y 674.038,Z 474.78,A -85,B 0,C 180,E1 4296.76,E2 4296.76} C_VEL
LIN {X 0,Y 674.458,Z 474.78,A -85,B 0,C 180,E1 4303.628,E2 4303.628} C_VEL
LIN {X 0,Y 674.566,Z 474.78,A -85,B 0,C 180,E1 4311.554,E2 4311.554} C_VEL
LIN {X 0,Y 675.148,Z 474.78,A -85,B 0,C 180,E1 4318.03,E2 4318.03} C_VEL
LIN {X 0,Y 675.018,Z 474.78,A -85,B 0,C 180,E1 4325.766,E2 4325.766} C_VEL
LIN {X 0,Y 674.71,Z 474.78,A -85,B 0,C 180,E1 4333.617,E2 4333.617} C_VEL
LIN {X 0,Y 674.445,Z 474.78,A -85,B 0,C 180,E1 4341.747,E2 4341.747} C_VEL
LIN {X 0,Y 674.648,Z 474.78,A -85,B 0,C 180,E1 4350.353,E2 4350.353} C_VEL
LIN {X 0,Y 674.395,Z 474.78,A -85,B 0,C 180,E1 4358.171,E2 4358.171} C_VEL
LIN {X 0,Y 674.21,Z 474.78,A -85,B 0,C 180,E1 4365.088,E2 4365.088} C_VEL
LIN {X 0,Y 674.647,Z 474.78,A -85,B 0,C 180,E1 4373.439,E2 4373.439} C_VEL
LIN {X 0,Y 674.461,Z 474.78,A -85,B 0,C 180,E1 4381.091,E2 4381.091} C_VEL
LIN {X 0,Y 674.281,Z 474.78,A -85,B 0,C 180,E1 4389.598,E2 4389.598} C_VEL
LIN {X 0,Y 674.513,Z 474.78,A -85,B 0,C 180,E1 4397.668,E2 4397.668} C_VEL
LIN {X 0,Y 675.391,Z 474.78,A -85,B 0,C 180,E1 4406.782,E2 4406.782} C_VEL
LIN {X 0,Y 674.951,Z 474.78,A -85,B 0,C 180,E1 4415.803,E2 4415.803} C_VEL
LIN {X 0,Y 674.732,Z 474.78,A -85,B 0,C 180,E1 4423.65,E2 4423.65} C_VEL
LIN {X 0,Y 674.435,Z 474.78,A -85,B 0,C 180,E1 4431.778,E2 4431.778} C_VEL
LIN {X 0,Y 674.265,Z 474.78,A -85,B 0,C 180,E1 4440.401,E2 4440.401} C_VEL
LIN {X 0,Y 674.186,Z 474.78,A -85,B 0,C 180,E1 4448.212,E2 4448.212} C_VEL
LIN {X 0,Y 674.315,Z 474.78,A -85,B 0,C 180,E1 4456.962,E2 4456.962} C_VEL
LIN {X 0,Y 674.222,Z 474.78,A -85,B 0,C 180,E1 4465.182,E2 4465.182} C_VEL
LIN {X 0,Y 674.331,Z 474.78,A -85,B 0,C 180,E1 4472.661,E2 4472.661} C_VEL
LIN {X 0,Y 674.493,Z 474.78,A -85,B 0,C 180,E1 4479.636,E2 4479.636} C_VEL
LIN {X 0,Y 675.369,Z 474.78,A -85,B 0,C 180,E1 4487.717,E2 4487.717} C_VEL
LIN {X 0,Y 675.12,Z 474.78,A -85,B 0,C 180,E1 4498.107,E2 4498.107} C_VEL
LIN {X 0,Y 674.99,Z 474.78,A -85,B 0,C 180,E1 4505.844,E2 4505.844} C_VEL
LIN {X 0,Y 674.715,Z 474.78,A -85,B 0,C 180,E1 4513.697,E2 4513.697} C_VEL
LIN {X 0,Y 674.393,Z 474.78,A -85,B 0,C 180,E1 4521.832,E2 4521.832} C_VEL
LIN {X 0,Y 674.427,Z 474.78,A -85,B 0,C 180,E1 4527.096,E2 4527.096} C_VEL
LIN {X 0,Y 666.289,Z 474.78,A -85,B 0,C 180,E1 4530.063,E2 4530.063} C_VEL
LIN {X 0,Y 666.119,Z 474.78,A -85,B 0,C 180,E1 4538.833,E2 4538.833} C_VEL
LIN {X 0,Y 666.434,Z 474.78,A -85,B 0,C 180,E1 4546.05,E2 4546.05} C_VEL
LIN {X 0,Y 666.517,Z 474.78,A -85,B 0,C 180,E1 4554.536,E2 4554.536} C_VEL
LIN {X 0,Y 666.578,Z 474.78,A -85,B 0,C 180,E1 4562.974,E2 4562.974} C_VEL
LIN {X 0,Y 667.097,Z 477.588,A -85,B 0,C 180,E1 4563.349,E2 4563.349} C_VEL
LIN {X 0,Y 676.15,Z 503.154,A -85,B 0,C 180,E1 4564.027,E2 4564.027} C_VEL
LIN {X 0,Y 675.103,Z 571.994,A -85,B 0,C 180,E1 4565.269,E2 4565.269} C_VEL
LIN {X 0,Y 672.864,Z 632.839,A -85,B 0,C 180,E1 4567.708,E2 4567.708} C_VEL
LIN {X 0,Y 670.538,Z 686.014,A -85,B 0,C 180,E1 4571.285,E2 4571.285} C_VEL
LIN {X 0,Y 668.668,Z 729.655,A -85,B 0,C 180,E1 4575.889,E2 4575.889} C_VEL
LIN {X 0,Y 667.915,Z 760.399,A -85,B 0,C 180,E1 4581.217,E2 4581.217} C_VEL
LIN {X 0,Y 667.412,Z 776.03,A -85,B 0,C 180,E1 4586.744,E2 4586.744} C_VEL
LIN {X 0,Y 667.652,Z 777.57,A -85,B 0,C 180,E1 4591.952,E2 4591.952} C_VEL
LIN {X 0,Y 667.131,Z 766.512,A -85,B 0,C 180,E1 4597.182,E2 4597.182} C_VEL
LIN {X 0,Y 667.892,Z 742.249,A -85,B 0,C 180,E1 4602.267,E2 4602.267} C_VEL
LIN {X 0,Y 669.428,Z 703.35,A -85,B 0,C 180,E1 4607.127,E2 4607.127} C_VEL
LIN {X 0,Y 671.899,Z 652.238,A -85,B 0,C 180,E1 4611.169,E2 4611.169} C_VEL
LIN {X 0,Y 674.311,Z 593.688,A -85,B 0,C 180,E1 4614.026,E2 4614.026} C_VEL
LIN {X 0,Y 676.088,Z 531.268,A -85,B 0,C 180,E1 4615.616,E2 4615.616} C_VEL
LIN {X 0,Y 674.125,Z 493.823,A -85,B 0,C 180,E1 4616.165,E2 4616.165} C_VEL
LIN {X 0,Y 667.221,Z 474.78,A -85,B 0,C 180,E1 4616.74,E2 4616.74} C_VEL
LIN {X 0,Y 666.57,Z 474.78,A -85,B 0,C 180,E1 4626.029,E2 4626.029} C_VEL
LIN {X 0,Y 666.286,Z 474.78,A -85,B 0,C 180,E1 4634.112,E2 4634.112} C_VEL
LIN {X 0,Y 666.609,Z 474.78,A -85,B 0,C 180,E1 4642.856,E2 4642.856} C_VEL
LIN {X 0,Y 666.483,Z 474.78,A -85,B 0,C 180,E1 4651.165,E2 4651.165} C_VEL
LIN {X 0,Y 666.169,Z 474.78,A -85,B 0,C 180,E1 4659.286,E2 4659.286} C_VEL
LIN {X 0,Y 666.151,Z 474.78,A -85,B 0,C 180,E1 4666.124,E2 4666.124} C_VEL
LIN {X 0,Y 666.251,Z 474.78,A -85,B 0,C 180,E1 4672.766,E2 4672.766} C_VEL
LIN {X 0,Y 666.546,Z 474.78,A -85,B 0,C 180,E1 4679.309,E2 4679.309} C_VEL
LIN {X 0,Y 666.968,Z 474.78,A -85,B 0,C 180,E1 4685.836,E2 4685.836} C_VEL
LIN {X 0,Y 666.632,Z 474.78,A -85,B 0,C 180,E1 4693.786,E2 4693.786} C_VEL
LIN {X 0,Y 666.325,Z 474.78,A -85,B 0,C 180,E1 4702.026,E2 4702.026} C_VEL
LIN {X 0,Y 666.577,Z 474.78,A -85,B 0,C 180,E1 4710.76,E2 4710.76} C_VEL
LIN {X 0,Y 666.38,Z 474.78,A -85,B 0,C 180,E1 4718.714,E2 4718.714} C_VEL
LIN {X 0,Y 666.093,Z 474.78,A -85,B 0,C 180,E1 4726.021,E2 4726.021} C_VEL
LIN {X 0,Y 666.643,Z 474.78,A -85,B 0,C 180,E1 4733.829,E2 4733.829} C_VEL
LIN {X 0,Y 666.574,Z 474.78,A -85,B 0,C 180,E1 4742.2,E2 4742.2} C_VEL
LIN {X 0,Y 666.791,Z 474.78,A -85,B 0,C 180,E1 4752.12,E2 4752.12} C_VEL
LIN {X 0,Y 666.958,Z 474.78,A -85,B 0,C 180,E1 4760.181,E2 4760.181} C_VEL
LIN {X 0,Y 667.055,Z 474.78,A -85,B 0,C 180,E1 4768.046,E2 4768.046} C_VEL
LIN {X 0,Y 666.904,Z 474.78,A -85,B 0,C 180,E1 4775.873,E2 4775.873} C_VEL
LIN {X 0,Y 666.651,Z 474.78,A -85,B 0,C 180,E1 4783.819,E2 4783.819} C_VEL
LIN {X 0,Y 666.315,Z 474.78,A -85,B 0,C 180,E1 4792.057,E2 4792.057} C_VEL
LIN {X 0,Y 666.469,Z 474.78,A -85,B 0,C 180,E1 4799.289,E2 4799.289} C_VEL
LIN {X 0,Y 666.167,Z 474.78,A -85,B 0,C 180,E1 4808.273,E2 4808.273} C_VEL
LIN {X 0,Y 666.371,Z 474.78,A -85,B 0,C 180,E1 4816.072,E2 4816.072} C_VEL
LIN {X 0,Y 666.254,Z 474.78,A -85,B 0,C 180,E1 4824.549,E2 4824.549} C_VEL
LIN {X 0,Y 666.377,Z 474.78,A -85,B 0,C 180,E1 4832.221,E2 4832.221} C_VEL
LIN {X 0,Y 666.548,Z 474.78,A -85,B 0,C 180,E1 4839.382,E2 4839.382} C_VEL
LIN {X 0,Y 667.365,Z 474.78,A -85,B 0,C 180,E1 4847.567,E2 4847.567} C_VEL
LIN {X 0,Y 667.124,Z 474.78,A -85,B 0,C 180,E1 4858.084,E2 4858.084} C_VEL
LIN {X 0,Y 666.941,Z 474.78,A -85,B 0,C 180,E1 4865.915,E2 4865.915} C_VEL
LIN {X 0,Y 666.632,Z 474.78,A -85,B 0,C 180,E1 4873.866,E2 4873.866} C_VEL
LIN {X 0,Y 666.278,Z 474.78,A -85,B 0,C 180,E1 4882.112,E2 4882.112} C_VEL
LIN {X 0,Y 666.289,Z 474.78,A -85,B 0,C 180,E1 4890.063,E2 4890.063} C_VEL
LIN {X 0,Y 657.974,Z 474.78,A -85,B 0,C 180,E1 4893.042,E2 4893.042} C_VEL
LIN {X 0,Y 657.992,Z 474.78,A -85,B 0,C 180,E1 4899.459,E2 4899.459} C_VEL
LIN {X 0,Y 658.24,Z 474.78,A -85,B 0,C 180,E1 4907.185,E2 4907.185} C_VEL
LIN {X 0,Y 658.437,Z 474.78,A -85,B 0,C 180,E1 4915.648,E2 4915.648} C_VEL
LIN {X 0,Y 658.689,Z 475.97,A -85,B 0,C 180,E1 4922.965,E2 4922.965} C_VEL
LIN {X 0,Y 668.967,Z 506.263,A -85,B 0,C 180,E1 4923.765,E2 4923.765} C_VEL
LIN {X 0,Y 667.735,Z 573.972,A -85,B 0,C 180,E1 4925.045,E2 4925.045} C_VEL
LIN {X 0,Y 665.303,Z 634.176,A -85,B 0,C 180,E1 4927.519,E2 4927.519} C_VEL
LIN {X 0,Y 662.779,Z 686.986,A -85,B 0,C 180,E1 4931.144,E2 4931.144} C_VEL
LIN {X 0,Y 660.742,Z 729.736,A -85,B 0,C 180,E1 4935.727,E2 4935.727} C_VEL
LIN {X 0,Y 659.926,Z 760.262,A -85,B 0,C 180,E1 4941.077,E2 4941.077} C_VEL
LIN {X 0,Y 659.425,Z 776.024,A -85,B 0,C 180,E1 4946.704,E2 4946.704} C_VEL
LIN {X 0,Y 659.655,Z 777.565,A -85,B 0,C 180,E1 4951.976,E2 4951.976} C_VEL
LIN {X 0,Y 659.178,Z 766.516,A -85,B 0,C 180,E1 4957.269,E2 4957.269} C_VEL
LIN {X 0,Y 660.081,Z 741.085,A -85,B 0,C 180,E1 4962.607,E2 4962.607} C_VEL
LIN {X 0,Y 661.753,Z 702.502,A -85,B 0,C 180,E1 4967.418,E2 4967.418} C_VEL
LIN {X 0,Y 664.371,Z 652.226,A -85,B 0,C 180,E1 4971.421,E2 4971.421} C_VEL
LIN {X 0,Y 666.94,Z 594.232,A -85,B 0,C 180,E1 4974.284,E2 4974.284} C_VEL
LIN {X 0,Y 668.869,Z 532.157,A -85,B 0,C 180,E1 4975.897,E2 4975.897} C_VEL
LIN {X 0,Y 667.056,Z 496.151,A -85,B 0,C 180,E1 4976.434,E2 4976.434} C_VEL
LIN {X 0,Y 659.143,Z 474.78,A -85,B 0,C 180,E1 4977.211,E2 4977.211} C_VEL
LIN {X 0,Y 658.607,Z 474.78,A -85,B 0,C 180,E1 4985.955,E2 4985.955} C_VEL
LIN {X 0,Y 658.172,Z 474.78,A -85,B 0,C 180,E1 4994.648,E2 4994.648} C_VEL
LIN {X 0,Y 658.61,Z 474.78,A -85,B 0,C 180,E1 5002.597,E2 5002.597} C_VEL
LIN {X 0,Y 658.402,Z 474.78,A -85,B 0,C 180,E1 5010.255,E2 5010.255} C_VEL
LIN {X 0,Y 657.995,Z 474.78,A -85,B 0,C 180,E1 5017.595,E2 5017.595} C_VEL
LIN {X 0,Y 658.216,Z 474.78,A -85,B 0,C 180,E1 5024.587,E2 5024.587} C_VEL
LIN {X 0,Y 658.62,Z 474.78,A -85,B 0,C 180,E1 5031.348,E2 5031.348} C_VEL
LIN {X 0,Y 659.16,Z 474.78,A -85,B 0,C 180,E1 5037.982,E2 5037.982} C_VEL
LIN {X 0,Y 658.92,Z 474.78,A -85,B 0,C 180,E1 5045.908,E2 5045.908} C_VEL
LIN {X 0,Y 658.578,Z 474.78,A -85,B 0,C 180,E1 5053.958,E2 5053.958} C_VEL
LIN {X 0,Y 658.259,Z 474.78,A -85,B 0,C 180,E1 5062.31,E2 5062.31} C_VEL
LIN {X 0,Y 658.557,Z 474.78,A -85,B 0,C 180,E1 5071.176,E2 5071.176} C_VEL
LIN {X 0,Y 658.367,Z 474.78,A -85,B 0,C 180,E1 5079.499,E2 5079.499} C_VEL
LIN {X 0,Y 658.129,Z 474.78,A -85,B 0,C 180,E1 5087.176,E2 5087.176} C_VEL
LIN {X 0,Y 658.72,Z 474.78,A -85,B 0,C 180,E1 5095.665,E2 5095.665} C_VEL
LIN {X 0,Y 658.454,Z 474.78,A -85,B 0,C 180,E1 5104.781,E2 5104.781} C_VEL
LIN {X 0,Y 658.547,Z 474.78,A -85,B 0,C 180,E1 5113.271,E2 5113.271} C_VEL
LIN {X 0,Y 658.559,Z 474.78,A -85,B 0,C 180,E1 5121.392,E2 5121.392} C_VEL
LIN {X 0,Y 659.084,Z 474.78,A -85,B 0,C 180,E1 5128.022,E2 5128.022} C_VEL
LIN {X 0,Y 658.859,Z 474.78,A -85,B 0,C 180,E1 5135.945,E2 5135.945} C_VEL
LIN {X 0,Y 658.589,Z 474.78,A -85,B 0,C 180,E1 5143.991,E2 5143.991} C_VEL
LIN {X 0,Y 658.242,Z 474.78,A -85,B 0,C 180,E1 5152.342,E2 5152.342} C_VEL
LIN {X 0,Y 658.201,Z 474.78,A -85,B 0,C 180,E1 5160.263,E2 5160.263} C_VEL
LIN {X 0,Y 658.256,Z 474.78,A -85,B 0,C 180,E1 5167.626,E2 5167.626} C_VEL
LIN {X 0,Y 658.275,Z 474.78,A -85,B 0,C 180,E1 5176.525,E2 5176.525} C_VEL
LIN {X 0,Y 658.196,Z 474.78,A -85,B 0,C 180,E1 5184.877,E2 5184.877} C_VEL
LIN {X 0,Y 658.335,Z 474.78,A -85,B 0,C 180,E1 5192.481,E2 5192.481} C_VEL
LIN {X 0,Y 658.341,Z 474.78,A -85,B 0,C 180,E1 5200.52,E2 5200.52} C_VEL
LIN {X 0,Y 659.329,Z 474.78,A -85,B 0,C 180,E1 5208.761,E2 5208.761} C_VEL
LIN {X 0,Y 659.134,Z 474.78,A -85,B 0,C 180,E1 5218.061,E2 5218.061} C_VEL
LIN {X 0,Y 658.895,Z 474.78,A -85,B 0,C 180,E1 5225.987,E2 5225.987} C_VEL
LIN {X 0,Y 658.583,Z 474.78,A -85,B 0,C 180,E1 5234.039,E2 5234.039} C_VEL
LIN {X 0,Y 658.202,Z 474.78,A -85,B 0,C 180,E1 5242.398,E2 5242.398} C_VEL
LIN {X 0,Y 658.277,Z 474.78,A -85,B 0,C 180,E1 5250.243,E2 5250.243} C_VEL
LIN {X 0,Y 657.974,Z 474.78,A -85,B 0,C 180,E1 5253.042,E2 5253.042} C_VEL
LIN {X 0,Y 650.266,Z 474.78,A -85,B 0,C 180,E1 5256.086,E2 5256.086} C_VEL
LIN {X 0,Y 650.409,Z 474.78,A -85,B 0,C 180,E1 5265.412,E2 5265.412} C_VEL
LIN {X 0,Y 650.537,Z 474.78,A -85,B 0,C 180,E1 5273.642,E2 5273.642} C_VEL
LIN {X 0,Y 650.546,Z 474.78,A -85,B 0,C 180,E1 5282.405,E2 5282.405} C_VEL
LIN {X 0,Y 661.774,Z 506.088,A -85,B 0,C 180,E1 5283.458,E2 5283.458} C_VEL
LIN {X 0,Y 660.456,Z 573.796,A -85,B 0,C 180,E1 5284.751,E2 5284.751} C_VEL
LIN {X 0,Y 657.852,Z 633.391,A -85,B 0,C 180,E1 5287.211,E2 5287.211} C_VEL
LIN {X 0,Y 655.058,Z 686.013,A -85,B 0,C 180,E1 5290.825,E2 5290.825} C_VEL
LIN {X 0,Y 652.831,Z 728.263,A -85,B 0,C 180,E1 5295.357,E2 5295.357} C_VEL
LIN {X 0,Y 651.923,Z 758.763,A -85,B 0,C 180,E1 5300.629,E2 5300.629} C_VEL
LIN {X 0,Y 651.602,Z 774.913,A -85,B 0,C 180,E1 5305.996,E2 5305.996} C_VEL
LIN {X 0,Y 651.652,Z 777.559,A -85,B 0,C 180,E1 5312,E2 5312} C_VEL
LIN {X 0,Y 651.207,Z 766.518,A -85,B 0,C 180,E1 5317.359,E2 5317.359} C_VEL
LIN {X 0,Y 652.172,Z 741.078,A -85,B 0,C 180,E1 5322.762,E2 5322.762} C_VEL
LIN {X 0,Y 653.992,Z 701.988,A -85,B 0,C 180,E1 5327.684,E2 5327.684} C_VEL
LIN {X 0,Y 656.825,Z 652.186,A -85,B 0,C 180,E1 5331.679,E2 5331.679} C_VEL
LIN {X 0,Y 659.608,Z 593.398,A -85,B 0,C 180,E1 5334.597,E2 5334.597} C_VEL
LIN {X 0,Y 661.672,Z 531.928,A -85,B 0,C 180,E1 5336.201,E2 5336.201} C_VEL
LIN {X 0,Y 659.796,Z 498.052,A -85,B 0,C 180,E1 5336.723,E2 5336.723} C_VEL
LIN {X 0,Y 651.127,Z 474.78,A -85,B 0,C 180,E1 5337.456,E2 5337.456} C_VEL
LIN {X 0,Y 650.516,Z 474.78,A -85,B 0,C 180,E1 5346.474,E2 5346.474} C_VEL
LIN {X 0,Y 650.182,Z 474.78,A -85,B 0,C 180,E1 5354.568,E2 5354.568} C_VEL
LIN {X 0,Y 650.596,Z 474.78,A -85,B 0,C 180,E1 5363.53,E2 5363.53} C_VEL
LIN {X 0,Y 650.469,Z 474.78,A -85,B 0,C 180,E1 5371.389,E2 5371.389} C_VEL
LIN {X 0,Y 650.525,Z 474.78,A -85,B 0,C 180,E1 5380.756,E2 5380.756} C_VEL
LIN {X 0,Y 650.887,Z 474.78,A -85,B 0,C 180,E1 5389.891,E2 5389.891} C_VEL
LIN {X 0,Y 651.161,Z 474.78,A -85,B 0,C 180,E1 5397.957,E2 5397.957} C_VEL
LIN {X 0,Y 650.876,Z 474.78,A -85,B 0,C 180,E1 5405.981,E2 5405.981} C_VEL
LIN {X 0,Y 650.361,Z 474.78,A -85,B 0,C 180,E1 5414.607,E2 5414.607} C_VEL
LIN {X 0,Y 650.158,Z 474.78,A -85,B 0,C 180,E1 5422.603,E2 5422.603} C_VEL
LIN {X 0,Y 650.51,Z 474.78,A -85,B 0,C 180,E1 5431.606,E2 5431.606} C_VEL
LIN {X 0,Y 650.38,Z 474.78,A -85,B 0,C 180,E1 5439.853,E2 5439.853} C_VEL
LIN {X 0,Y 650.289,Z 474.78,A -85,B 0,C 180,E1 5448.346,E2 5448.346} C_VEL
LIN {X 0,Y 650.655,Z 474.78,A -85,B 0,C 180,E1 5456.79,E2 5456.79} C_VEL
LIN {X 0,Y 650.45,Z 474.78,A -85,B 0,C 180,E1 5464.449,E2 5464.449} C_VEL
LIN {X 0,Y 650.605,Z 474.78,A -85,B 0,C 180,E1 5473.061,E2 5473.061} C_VEL
LIN {X 0,Y 650.6,Z 474.78,A -85,B 0,C 180,E1 5481.286,E2 5481.286} C_VEL
LIN {X 0,Y 651.086,Z 474.78,A -85,B 0,C 180,E1 5487.998,E2 5487.998} C_VEL
LIN {X 0,Y 650.817,Z 474.78,A -85,B 0,C 180,E1 5496.019,E2 5496.019} C_VEL
LIN {X 0,Y 650.362,Z 474.78,A -85,B 0,C 180,E1 5504.66,E2 5504.66} C_VEL
LIN {X 0,Y 650.141,Z 474.78,A -85,B 0,C 180,E1 5512.636,E2 5512.636} C_VEL
LIN {X 0,Y 650.244,Z 474.78,A -85,B 0,C 180,E1 5520.094,E2 5520.094} C_VEL
LIN {X 0,Y 649.999,Z 474.78,A -85,B 0,C 180,E1 5528.625,E2 5528.625} C_VEL
LIN {X 0,Y 650.165,Z 474.78,A -85,B 0,C 180,E1 5537.284,E2 5537.284} C_VEL
LIN {X 0,Y 650.155,Z 474.78,A -85,B 0,C 180,E1 5545.177,E2 5545.177} C_VEL
LIN {X 0,Y 650.249,Z 474.78,A -85,B 0,C 180,E1 5552.981,E2 5552.981} C_VEL
LIN {X 0,Y 650.312,Z 474.78,A -85,B 0,C 180,E1 5560.81,E2 5560.81} C_VEL
LIN {X 0,Y 651.322,Z 474.78,A -85,B 0,C 180,E1 5568.621,E2 5568.621} C_VEL
LIN {X 0,Y 651.137,Z 474.78,A -85,B 0,C 180,E1 5578.037,E2 5578.037} C_VEL
LIN {X 0,Y 650.85,Z 474.78,A -85,B 0,C 180,E1 5586.062,E2 5586.062} C_VEL
LIN {X 0,Y 650.385,Z 474.78,A -85,B 0,C 180,E1 5594.614,E2 5594.614} C_VEL
LIN {X 0,Y 650.096,Z 474.78,A -85,B 0,C 180,E1 5602.865,E2 5602.865} C_VEL
LIN {X 0,Y 650.322,Z 474.78,A -85,B 0,C 180,E1 5610.152,E2 5610.152} C_VEL
LIN {X 0,Y 650.266,Z 474.78,A -85,B 0,C 180,E1 5616.086,E2 5616.086} C_VEL
LIN {X 0,Y 641.98,Z 474.78,A -85,B 0,C 180,E1 5619.151,E2 5619.151} C_VEL
LIN {X 0,Y 642.199,Z 474.78,A -85,B 0,C 180,E1 5627.701,E2 5627.701} C_VEL
LIN {X 0,Y 642.428,Z 474.78,A -85,B 0,C 180,E1 5636.308,E2 5636.308} C_VEL
LIN {X 0,Y 642.551,Z 474.869,A -85,B 0,C 180,E1 5642.219,E2 5642.219} C_VEL
LIN {X 0,Y 654.604,Z 510.327,A -85,B 0,C 180,E1 5643.197,E2 5643.197} C_VEL
LIN {X 0,Y 652.985,Z 577.108,A -85,B 0,C 180,E1 5644.555,E2 5644.555} C_VEL
LIN {X 0,Y 650.084,Z 637.869,A -85,B 0,C 180,E1 5647.199,E2 5647.199} C_VEL
LIN {X 0,Y 647.148,Z 690.75,A -85,B 0,C 180,E1 5651.026,E2 5651.026} C_VEL
LIN {X 0,Y 644.912,Z 732.043,A -85,B 0,C 180,E1 5655.706,E2 5655.706} C_VEL
LIN {X 0,Y 643.931,Z 761.601,A -85,B 0,C 180,E1 5661.195,E2 5661.195} C_VEL
LIN {X 0,Y 643.446,Z 776.014,A -85,B 0,C 180,E1 5666.622,E2 5666.622} C_VEL
LIN {X 0,Y 643.678,Z 777.553,A -85,B 0,C 180,E1 5672.025,E2 5672.025} C_VEL
LIN {X 0,Y 643.247,Z 766.518,A -85,B 0,C 180,E1 5677.45,E2 5677.45} C_VEL
LIN {X 0,Y 644.295,Z 741.071,A -85,B 0,C 180,E1 5682.921,E2 5682.921} C_VEL
LIN {X 0,Y 646.288,Z 701.781,A -85,B 0,C 180,E1 5687.923,E2 5687.923} C_VEL
LIN {X 0,Y 649.256,Z 652.007,A -85,B 0,C 180,E1 5691.945,E2 5691.945} C_VEL
LIN {X 0,Y 652.295,Z 593.222,A -85,B 0,C 180,E1 5694.891,E2 5694.891} C_VEL
LIN {X 0,Y 654.509,Z 531.753,A -85,B 0,C 180,E1 5696.51,E2 5696.51} C_VEL
LIN {X 0,Y 652.79,Z 500.355,A -85,B 0,C 180,E1 5697.003,E2 5697.003} C_VEL
LIN {X 0,Y 643.091,Z 474.78,A -85,B 0,C 180,E1 5697.798,E2 5697.798} C_VEL
LIN {X 0,Y 642.383,Z 474.78,A -85,B 0,C 180,E1 5707.012,E2 5707.012} C_VEL
LIN {X 0,Y 642.232,Z 474.78,A -85,B 0,C 180,E1 5714.153,E2 5714.153} C_VEL
LIN {X 0,Y 642.51,Z 474.78,A -85,B 0,C 180,E1 5722.925,E2 5722.925} C_VEL
LIN {X 0,Y 642.444,Z 474.78,A -85,B 0,C 180,E1 5730.998,E2 5730.998} C_VEL
LIN {X 0,Y 642.313,Z 474.78,A -85,B 0,C 180,E1 5739.927,E2 5739.927} C_VEL
LIN {X 0,Y 642.713,Z 474.78,A -85,B 0,C 180,E1 5748.383,E2 5748.383} C_VEL
LIN {X 0,Y 643.185,Z 474.78,A -85,B 0,C 180,E1 5757.932,E2 5757.932} C_VEL
LIN {X 0,Y 642.85,Z 474.78,A -85,B 0,C 180,E1 5766.056,E2 5766.056} C_VEL
LIN {X 0,Y 642.467,Z 474.78,A -85,B 0,C 180,E1 5774.315,E2 5774.315} C_VEL
LIN {X 0,Y 642.098,Z 474.78,A -85,B 0,C 180,E1 5782.903,E2 5782.903} C_VEL
LIN {X 0,Y 642.552,Z 474.78,A -85,B 0,C 180,E1 5790.522,E2 5790.522} C_VEL
LIN {X 0,Y 642.36,Z 474.78,A -85,B 0,C 180,E1 5798.697,E2 5798.697} C_VEL
LIN {X 0,Y 642.1,Z 474.78,A -85,B 0,C 180,E1 5806.052,E2 5806.052} C_VEL
LIN {X 0,Y 642.62,Z 474.78,A -85,B 0,C 180,E1 5814.679,E2 5814.679} C_VEL
LIN {X 0,Y 642.492,Z 474.78,A -85,B 0,C 180,E1 5822.596,E2 5822.596} C_VEL
LIN {X 0,Y 642.657,Z 474.78,A -85,B 0,C 180,E1 5831.424,E2 5831.424} C_VEL
LIN {X 0,Y 642.614,Z 474.78,A -85,B 0,C 180,E1 5841.177,E2 5841.177} C_VEL
LIN {X 0,Y 643.099,Z 474.78,A -85,B 0,C 180,E1 5847.973,E2 5847.973} C_VEL
LIN {X 0,Y 642.791,Z 474.78,A -85,B 0,C 180,E1 5856.094,E2 5856.094} C_VEL
LIN {X 0,Y 642.474,Z 474.78,A -85,B 0,C 180,E1 5864.35,E2 5864.35} C_VEL
LIN {X 0,Y 642.082,Z 474.78,A -85,B 0,C 180,E1 5872.936,E2 5872.936} C_VEL
LIN {X 0,Y 642.151,Z 474.78,A -85,B 0,C 180,E1 5880.513,E2 5880.513} C_VEL
LIN {X 0,Y 641.982,Z 474.78,A -85,B 0,C 180,E1 5888.754,E2 5888.754} C_VEL
LIN {X 0,Y 642.282,Z 474.78,A -85,B 0,C 180,E1 5896.066,E2 5896.066} C_VEL
LIN {X 0,Y 642.154,Z 474.78,A -85,B 0,C 180,E1 5904.679,E2 5904.679} C_VEL
LIN {X 0,Y 642.246,Z 474.78,A -85,B 0,C 180,E1 5912.616,E2 5912.616} C_VEL
LIN {X 0,Y 642.372,Z 474.78,A -85,B 0,C 180,E1 5920.015,E2 5920.015} C_VEL
LIN {X 0,Y 643.304,Z 474.78,A -85,B 0,C 180,E1 5928.477,E2 5928.477} C_VEL
LIN {X 0,Y 643.162,Z 474.78,A -85,B 0,C 180,E1 5938.013,E2 5938.013} C_VEL
LIN {X 0,Y 642.83,Z 474.78,A -85,B 0,C 180,E1 5946.138,E2 5946.138} C_VEL
LIN {X 0,Y 642.455,Z 474.78,A -85,B 0,C 180,E1 5954.399,E2 5954.399} C_VEL
LIN {X 0,Y 642.067,Z 474.78,A -85,B 0,C 180,E1 5962.992,E2 5962.992} C_VEL
LIN {X 0,Y 642.237,Z 474.78,A -85,B 0,C 180,E1 5970.572,E2 5970.572} C_VEL
LIN {X 0,Y 641.98,Z 474.78,A -85,B 0,C 180,E1 5979.151,E2 5979.151} C_VEL
LIN {X 0,Y 633.972,Z 474.78,A -85,B 0,C 180,E1 5982.267,E2 5982.267} C_VEL
LIN {X 0,Y 634.311,Z 474.78,A -85,B 0,C 180,E1 5991.086,E2 5991.086} C_VEL
LIN {X 0,Y 634.551,Z 474.78,A -85,B 0,C 180,E1 5999.081,E2 5999.081} C_VEL
LIN {X 0,Y 634.703,Z 476.349,A -85,B 0,C 180,E1 6001.866,E2 6001.866} C_VEL
LIN {X 0,Y 647.411,Z 513.454,A -85,B 0,C 180,E1 6002.915,E2 6002.915} C_VEL
LIN {X 0,Y 645.62,Z 578.909,A -85,B 0,C 180,E1 6004.309,E2 6004.309} C_VEL
LIN {X 0,Y 642.53,Z 638.91,A -85,B 0,C 180,E1 6006.989,E2 6006.989} C_VEL
LIN {X 0,Y 639.412,Z 690.576,A -85,B 0,C 180,E1 6010.787,E2 6010.787} C_VEL
LIN {X 0,Y 637.009,Z 732.035,A -85,B 0,C 180,E1 6015.524,E2 6015.524} C_VEL
LIN {X 0,Y 635.97,Z 761.594,A -85,B 0,C 180,E1 6021.083,E2 6021.083} C_VEL
LIN {X 0,Y 635.454,Z 776.009,A -85,B 0,C 180,E1 6026.58,E2 6026.58} C_VEL
LIN {X 0,Y 635.675,Z 777.547,A -85,B 0,C 180,E1 6032.051,E2 6032.051} C_VEL
LIN {X 0,Y 635.308,Z 766.515,A -85,B 0,C 180,E1 6037.544,E2 6037.544} C_VEL
LIN {X 0,Y 636.404,Z 741.064,A -85,B 0,C 180,E1 6043.084,E2 6043.084} C_VEL
LIN {X 0,Y 638.438,Z 703.059,A -85,B 0,C 180,E1 6048.003,E2 6048.003} C_VEL
LIN {X 0,Y 641.643,Z 652.966,A -85,B 0,C 180,E1 6052.142,E2 6052.142} C_VEL
LIN {X 0,Y 644.909,Z 594.431,A -85,B 0,C 180,E1 6055.142,E2 6055.142} C_VEL
LIN {X 0,Y 647.329,Z 532.262,A -85,B 0,C 180,E1 6056.817,E2 6056.817} C_VEL
LIN {X 0,Y 645.211,Z 501.298,A -85,B 0,C 180,E1 6057.333,E2 6057.333} C_VEL
LIN {X 0,Y 634.984,Z 474.78,A -85,B 0,C 180,E1 6058.309,E2 6058.309} C_VEL
LIN {X 0,Y 634.331,Z 474.78,A -85,B 0,C 180,E1 6067.562,E2 6067.562} C_VEL
LIN {X 0,Y 634.068,Z 474.78,A -85,B 0,C 180,E1 6075.041,E2 6075.041} C_VEL
LIN {X 0,Y 634.52,Z 474.78,A -85,B 0,C 180,E1 6084.088,E2 6084.088} C_VEL
LIN {X 0,Y 634.49,Z 474.78,A -85,B 0,C 180,E1 6092.16,E2 6092.16} C_VEL
LIN {X 0,Y 634.535,Z 474.78,A -85,B 0,C 180,E1 6101.125,E2 6101.125} C_VEL
LIN {X 0,Y 634.656,Z 474.78,A -85,B 0,C 180,E1 6111.019,E2 6111.019} C_VEL
LIN {X 0,Y 635.184,Z 474.78,A -85,B 0,C 180,E1 6117.906,E2 6117.906} C_VEL
LIN {X 0,Y 634.807,Z 474.78,A -85,B 0,C 180,E1 6126.133,E2 6126.133} C_VEL
LIN {X 0,Y 634.407,Z 474.78,A -85,B 0,C 180,E1 6134.508,E2 6134.508} C_VEL
LIN {X 0,Y 634.086,Z 474.78,A -85,B 0,C 180,E1 6142.961,E2 6142.961} C_VEL
LIN {X 0,Y 634.52,Z 474.78,A -85,B 0,C 180,E1 6150.889,E2 6150.889} C_VEL
LIN {X 0,Y 634.346,Z 474.78,A -85,B 0,C 180,E1 6159.28,E2 6159.28} C_VEL
LIN {X 0,Y 634.081,Z 474.78,A -85,B 0,C 180,E1 6167.03,E2 6167.03} C_VEL
LIN {X 0,Y 634.588,Z 474.78,A -85,B 0,C 180,E1 6175.501,E2 6175.501} C_VEL
LIN {X 0,Y 634.446,Z 474.78,A -85,B 0,C 180,E1 6183.756,E2 6183.756} C_VEL
LIN {X 0,Y 634.594,Z 474.78,A -85,B 0,C 180,E1 6192.62,E2 6192.62} C_VEL
LIN {X 0,Y 634.643,Z 474.78,A -85,B 0,C 180,E1 6201.065,E2 6201.065} C_VEL
LIN {X 0,Y 635.1,Z 474.78,A -85,B 0,C 180,E1 6207.947,E2 6207.947} C_VEL
LIN {X 0,Y 634.75,Z 474.78,A -85,B 0,C 180,E1 6216.172,E2 6216.172} C_VEL
LIN {X 0,Y 634.424,Z 474.78,A -85,B 0,C 180,E1 6224.572,E2 6224.572} C_VEL
LIN {X 0,Y 634.091,Z 474.78,A -85,B 0,C 180,E1 6233.002,E2 6233.002} C_VEL
LIN {X 0,Y 634.037,Z 474.78,A -85,B 0,C 180,E1 6240.946,E2 6240.946} C_VEL
LIN {X 0,Y 633.892,Z 474.78,A -85,B 0,C 180,E1 6249.344,E2 6249.344} C_VEL
LIN {X 0,Y 634.126,Z 474.78,A -85,B 0,C 180,E1 6257.064,E2 6257.064} C_VEL
LIN {X 0,Y 634.077,Z 474.78,A -85,B 0,C 180,E1 6265.834,E2 6265.834} C_VEL
LIN {X 0,Y 634.21,Z 474.78,A -85,B 0,C 180,E1 6273.778,E2 6273.778} C_VEL
LIN {X 0,Y 634.277,Z 474.78,A -85,B 0,C 180,E1 6281.203,E2 6281.203} C_VEL
LIN {X 0,Y 635.315,Z 474.78,A -85,B 0,C 180,E1 6288.33,E2 6288.33} C_VEL
LIN {X 0,Y 635.164,Z 474.78,A -85,B 0,C 180,E1 6297.988,E2 6297.988} C_VEL
LIN {X 0,Y 634.787,Z 474.78,A -85,B 0,C 180,E1 6306.216,E2 6306.216} C_VEL
LIN {X 0,Y 634.402,Z 474.78,A -85,B 0,C 180,E1 6314.586,E2 6314.586} C_VEL
LIN {X 0,Y 634.081,Z 474.78,A -85,B 0,C 180,E1 6322.96,E2 6322.96} C_VEL
LIN {X 0,Y 634.117,Z 474.78,A -85,B 0,C 180,E1 6331.006,E2 6331.006} C_VEL
LIN {X 0,Y 633.95,Z 474.78,A -85,B 0,C 180,E1 6339.415,E2 6339.415} C_VEL
LIN {X 0,Y 633.972,Z 474.78,A -85,B 0,C 180,E1 6342.267,E2 6342.267} C_VEL
LIN {X 0,Y 626.179,Z 474.78,A -85,B 0,C 180,E1 6345.428,E2 6345.428} C_VEL
LIN {X 0,Y 626.39,Z 474.78,A -85,B 0,C 180,E1 6354.306,E2 6354.306} C_VEL
LIN {X 0,Y 626.557,Z 475.32,A -85,B 0,C 180,E1 6361.457,E2 6361.457} C_VEL
LIN {X 0,Y 640.301,Z 515.889,A -85,B 0,C 180,E1 6362.622,E2 6362.622} C_VEL
LIN {X 0,Y 638.236,Z 581.609,A -85,B 0,C 180,E1 6364.086,E2 6364.086} C_VEL
LIN {X 0,Y 634.848,Z 641.495,A -85,B 0,C 180,E1 6366.863,E2 6366.863} C_VEL
LIN {X 0,Y 631.601,Z 692.294,A -85,B 0,C 180,E1 6370.723,E2 6370.723} C_VEL
LIN {X 0,Y 629.087,Z 734.311,A -85,B 0,C 180,E1 6375.695,E2 6375.695} C_VEL
LIN {X 0,Y 627.883,Z 762.839,A -85,B 0,C 180,E1 6381.318,E2 6381.318} C_VEL
LIN {X 0,Y 627.462,Z 776.004,A -85,B 0,C 180,E1 6386.536,E2 6386.536} C_VEL
LIN {X 0,Y 627.672,Z 777.541,A -85,B 0,C 180,E1 6392.077,E2 6392.077} C_VEL
LIN {X 0,Y 627.338,Z 766.509,A -85,B 0,C 180,E1 6397.64,E2 6397.64} C_VEL
LIN {X 0,Y 628.52,Z 741.057,A -85,B 0,C 180,E1 6403.251,E2 6403.251} C_VEL
LIN {X 0,Y 630.832,Z 701.503,A -85,B 0,C 180,E1 6408.376,E2 6408.376} C_VEL
LIN {X 0,Y 634.258,Z 650.871,A -85,B 0,C 180,E1 6412.546,E2 6412.546} C_VEL
LIN {X 0,Y 637.808,Z 591.648,A -85,B 0,C 180,E1 6415.546,E2 6415.546} C_VEL
LIN {X 0,Y 640.256,Z 529.523,A -85,B 0,C 180,E1 6417.177,E2 6417.177} C_VEL
LIN {X 0,Y 638.346,Z 504.031,A -85,B 0,C 180,E1 6417.616,E2 6417.616} C_VEL
LIN {X 0,Y 626.926,Z 474.78,A -85,B 0,C 180,E1 6418.609,E2 6418.609} C_VEL
LIN {X 0,Y 626.284,Z 474.78,A -85,B 0,C 180,E1 6428.131,E2 6428.131} C_VEL
LIN {X 0,Y 625.983,Z 474.78,A -85,B 0,C 180,E1 6436.252,E2 6436.252} C_VEL
LIN {X 0,Y 626.543,Z 474.78,A -85,B 0,C 180,E1 6445.264,E2 6445.264} C_VEL
LIN {X 0,Y 626.459,Z 474.78,A -85,B 0,C 180,E1 6453.335,E2 6453.335} C_VEL
LIN {X 0,Y 626.446,Z 474.78,A -85,B 0,C 180,E1 6462.981,E2 6462.981} C_VEL
LIN {X 0,Y 626.659,Z 474.78,A -85,B 0,C 180,E1 6470.904,E2 6470.904} C_VEL
LIN {X 0,Y 627.202,Z 474.78,A -85,B 0,C 180,E1 6477.879,E2 6477.879} C_VEL
LIN {X 0,Y 626.775,Z 474.78,A -85,B 0,C 180,E1 6486.212,E2 6486.212} C_VEL
LIN {X 0,Y 626.374,Z 474.78,A -85,B 0,C 180,E1 6494.691,E2 6494.691} C_VEL
LIN {X 0,Y 626.249,Z 474.78,A -85,B 0,C 180,E1 6502.012,E2 6502.012} C_VEL
LIN {X 0,Y 626.513,Z 474.78,A -85,B 0,C 180,E1 6511.328,E2 6511.328} C_VEL
LIN {X 0,Y 626.297,Z 474.78,A -85,B 0,C 180,E1 6519.884,E2 6519.884} C_VEL
LIN {X 0,Y 626.171,Z 474.78,A -85,B 0,C 180,E1 6528.24,E2 6528.24} C_VEL
LIN {X 0,Y 626.532,Z 474.78,A -85,B 0,C 180,E1 6537.003,E2 6537.003} C_VEL
LIN {X 0,Y 626.291,Z 474.78,A -85,B 0,C 180,E1 6545.193,E2 6545.193} C_VEL
LIN {X 0,Y 626.363,Z 474.78,A -85,B 0,C 180,E1 6553.834,E2 6553.834} C_VEL
LIN {X 0,Y 626.65,Z 474.78,A -85,B 0,C 180,E1 6560.95,E2 6560.95} C_VEL
LIN {X 0,Y 627.112,Z 474.78,A -85,B 0,C 180,E1 6567.921,E2 6567.921} C_VEL
LIN {X 0,Y 626.719,Z 474.78,A -85,B 0,C 180,E1 6576.251,E2 6576.251} C_VEL
LIN {X 0,Y 626.399,Z 474.78,A -85,B 0,C 180,E1 6584.726,E2 6584.726} C_VEL
LIN {X 0,Y 626.237,Z 474.78,A -85,B 0,C 180,E1 6592.046,E2 6592.046} C_VEL
LIN {X 0,Y 626.063,Z 474.78,A -85,B 0,C 180,E1 6600.73,E2 6600.73} C_VEL
LIN {X 0,Y 626.012,Z 474.78,A -85,B 0,C 180,E1 6608.15,E2 6608.15} C_VEL
LIN {X 0,Y 626.138,Z 474.78,A -85,B 0,C 180,E1 6616.381,E2 6616.381} C_VEL
LIN {X 0,Y 626.072,Z 474.78,A -85,B 0,C 180,E1 6625.336,E2 6625.336} C_VEL
LIN {X 0,Y 626.198,Z 474.78,A -85,B 0,C 180,E1 6633.416,E2 6633.416} C_VEL
LIN {X 0,Y 626.317,Z 474.78,A -85,B 0,C 180,E1 6640.955,E2 6640.955} C_VEL
LIN {X 0,Y 627.311,Z 474.78,A -85,B 0,C 180,E1 6648.255,E2 6648.255} C_VEL
LIN {X 0,Y 627.184,Z 474.78,A -85,B 0,C 180,E1 6657.962,E2 6657.962} C_VEL
LIN {X 0,Y 626.76,Z 474.78,A -85,B 0,C 180,E1 6666.296,E2 6666.296} C_VEL
LIN {X 0,Y 626.34,Z 474.78,A -85,B 0,C 180,E1 6674.778,E2 6674.778} C_VEL
LIN {X 0,Y 626.226,Z 474.78,A -85,B 0,C 180,E1 6682.102,E2 6682.102} C_VEL
LIN {X 0,Y 626.123,Z 474.78,A -85,B 0,C 180,E1 6690.704,E2 6690.704} C_VEL
LIN {X 0,Y 626.062,Z 474.78,A -85,B 0,C 180,E1 6698.221,E2 6698.221} C_VEL
LIN {X 0,Y 626.179,Z 474.78,A -85,B 0,C 180,E1 6705.428,E2 6705.428} C_VEL
LIN {X 0,Y 618.064,Z 474.78,A -85,B 0,C 180,E1 6708.619,E2 6708.619} C_VEL
LIN {X 0,Y 618.355,Z 474.78,A -85,B 0,C 180,E1 6716.509,E2 6716.509} C_VEL
LIN {X 0,Y 618.69,Z 476.191,A -85,B 0,C 180,E1 6721.074,E2 6721.074} C_VEL
LIN {X 0,Y 633.201,Z 516.225,A -85,B 0,C 180,E1 6722.295,E2 6722.295} C_VEL
LIN {X 0,Y 630.995,Z 581.633,A -85,B 0,C 180,E1 6723.773,E2 6723.773} C_VEL
LIN {X 0,Y 627.41,Z 641.535,A -85,B 0,C 180,E1 6726.585,E2 6726.585} C_VEL
LIN {X 0,Y 623.837,Z 692.161,A -85,B 0,C 180,E1 6730.478,E2 6730.478} C_VEL
LIN {X 0,Y 621.163,Z 734.132,A -85,B 0,C 180,E1 6735.508,E2 6735.508} C_VEL
LIN {X 0,Y 619.938,Z 762.832,A -85,B 0,C 180,E1 6741.206,E2 6741.206} C_VEL
LIN {X 0,Y 619.47,Z 775.999,A -85,B 0,C 180,E1 6746.491,E2 6746.491} C_VEL
LIN {X 0,Y 619.669,Z 777.535,A -85,B 0,C 180,E1 6752.104,E2 6752.104} C_VEL
LIN {X 0,Y 619.376,Z 766.504,A -85,B 0,C 180,E1 6757.739,E2 6757.739} C_VEL
LIN {X 0,Y 620.637,Z 740.882,A -85,B 0,C 180,E1 6763.422,E2 6763.422} C_VEL
LIN {X 0,Y 623.053,Z 701.843,A -85,B 0,C 180,E1 6768.557,E2 6768.557} C_VEL
LIN {X 0,Y 626.704,Z 651.298,A -85,B 0,C 180,E1 6772.79,E2 6772.79} C_VEL
LIN {X 0,Y 630.504,Z 591.817,A -85,B 0,C 180,E1 6775.849,E2 6775.849} C_VEL
LIN {X 0,Y 633.153,Z 529.349,A -85,B 0,C 180,E1 6777.507,E2 6777.507} C_VEL
LIN {X 0,Y 630.93,Z 505.34,A -85,B 0,C 180,E1 6777.95,E2 6777.95} C_VEL
LIN {X 0,Y 618.789,Z 474.78,A -85,B 0,C 180,E1 6779.138,E2 6779.138} C_VEL
LIN {X 0,Y 618.29,Z 474.78,A -85,B 0,C 180,E1 6787.037,E2 6787.037} C_VEL
LIN {X 0,Y 618.015,Z 474.78,A -85,B 0,C 180,E1 6795.541,E2 6795.541} C_VEL
LIN {X 0,Y 618.516,Z 474.78,A -85,B 0,C 180,E1 6804.747,E2 6804.747} C_VEL
LIN {X 0,Y 618.441,Z 474.78,A -85,B 0,C 180,E1 6813.511,E2 6813.511} C_VEL
LIN {X 0,Y 618.512,Z 474.78,A -85,B 0,C 180,E1 6822.1,E2 6822.1} C_VEL
LIN {X 0,Y 618.66,Z 474.78,A -85,B 0,C 180,E1 6830.785,E2 6830.785} C_VEL
LIN {X 0,Y 619.199,Z 474.78,A -85,B 0,C 180,E1 6837.852,E2 6837.852} C_VEL
LIN {X 0,Y 618.541,Z 474.78,A -85,B 0,C 180,E1 6846.81,E2 6846.81} C_VEL
LIN {X 0,Y 618.331,Z 474.78,A -85,B 0,C 180,E1 6854.887,E2 6854.887} C_VEL
LIN {X 0,Y 618.014,Z 474.78,A -85,B 0,C 180,E1 6863.048,E2 6863.048} C_VEL
LIN {X 0,Y 618.451,Z 474.78,A -85,B 0,C 180,E1 6871.784,E2 6871.784} C_VEL
LIN {X 0,Y 618.298,Z 474.78,A -85,B 0,C 180,E1 6880.507,E2 6880.507} C_VEL
LIN {X 0,Y 618.293,Z 474.78,A -85,B 0,C 180,E1 6889.461,E2 6889.461} C_VEL
LIN {X 0,Y 618.406,Z 474.78,A -85,B 0,C 180,E1 6898.181,E2 6898.181} C_VEL
LIN {X 0,Y 618.106,Z 474.78,A -85,B 0,C 180,E1 6906.12,E2 6906.12} C_VEL
LIN {X 0,Y 618.414,Z 474.78,A -85,B 0,C 180,E1 6913.62,E2 6913.62} C_VEL
LIN {X 0,Y 618.377,Z 474.78,A -85,B 0,C 180,E1 6922.248,E2 6922.248} C_VEL
LIN {X 0,Y 618.514,Z 474.78,A -85,B 0,C 180,E1 6929.298,E2 6929.298} C_VEL
LIN {X 0,Y 618.494,Z 474.78,A -85,B 0,C 180,E1 6936.898,E2 6936.898} C_VEL
LIN {X 0,Y 618.367,Z 474.78,A -85,B 0,C 180,E1 6944.922,E2 6944.922} C_VEL
LIN {X 0,Y 618.031,Z 474.78,A -85,B 0,C 180,E1 6953.095,E2 6953.095} C_VEL
LIN {X 0,Y 617.906,Z 474.78,A -85,B 0,C 180,E1 6961.848,E2 6961.848} C_VEL
LIN {X 0,Y 617.784,Z 474.78,A -85,B 0,C 180,E1 6970.579,E2 6970.579} C_VEL
LIN {X 0,Y 618.033,Z 474.78,A -85,B 0,C 180,E1 6978.451,E2 6978.451} C_VEL
LIN {X 0,Y 618.073,Z 474.78,A -85,B 0,C 180,E1 6986.524,E2 6986.524} C_VEL
LIN {X 0,Y 618.21,Z 474.78,A -85,B 0,C 180,E1 6994.612,E2 6994.612} C_VEL
LIN {X 0,Y 618.6,Z 474.78,A -85,B 0,C 180,E1 7003.661,E2 7003.661} C_VEL
LIN {X 0,Y 618.789,Z 474.78,A -85,B 0,C 180,E1 7010.872,E2 7010.872} C_VEL
LIN {X 0,Y 619.184,Z 474.78,A -85,B 0,C 180,E1 7017.936,E2 7017.936} C_VEL
LIN {X 0,Y 618.564,Z 474.78,A -85,B 0,C 180,E1 7026.827,E2 7026.827} C_VEL
LIN {X 0,Y 618.292,Z 474.78,A -85,B 0,C 180,E1 7034.975,E2 7034.975} C_VEL
LIN {X 0,Y 618.001,Z 474.78,A -85,B 0,C 180,E1 7043.045,E2 7043.045} C_VEL
LIN {X 0,Y 618.162,Z 474.78,A -85,B 0,C 180,E1 7050.257,E2 7050.257} C_VEL
LIN {X 0,Y 617.882,Z 474.78,A -85,B 0,C 180,E1 7059.366,E2 7059.366} C_VEL
LIN {X 0,Y 618.11,Z 474.78,A -85,B 0,C 180,E1 7067.57,E2 7067.57} C_VEL
LIN {X 0,Y 618.064,Z 474.78,A -85,B 0,C 180,E1 7068.619,E2 7068.619} C_VEL
LIN {X 0,Y 610.202,Z 474.78,A -85,B 0,C 180,E1 7071.859,E2 7071.859} C_VEL
LIN {X 0,Y 610.674,Z 476.244,A -85,B 0,C 180,E1 7080.661,E2 7080.661} C_VEL
LIN {X 0,Y 626.105,Z 517.462,A -85,B 0,C 180,E1 7081.972,E2 7081.972} C_VEL
LIN {X 0,Y 623.677,Z 583.429,A -85,B 0,C 180,E1 7083.51,E2 7083.51} C_VEL
LIN {X 0,Y 619.833,Z 643.266,A -85,B 0,C 180,E1 7086.401,E2 7086.401} C_VEL
LIN {X 0,Y 616.014,Z 694.036,A -85,B 0,C 180,E1 7090.422,E2 7090.422} C_VEL
LIN {X 0,Y 613.226,Z 735.127,A -85,B 0,C 180,E1 7095.499,E2 7095.499} C_VEL
LIN {X 0,Y 611.972,Z 762.677,A -85,B 0,C 180,E1 7101.09,E2 7101.09} C_VEL
LIN {X 0,Y 611.495,Z 775.965,A -85,B 0,C 180,E1 7106.445,E2 7106.445} C_VEL
LIN {X 0,Y 611.666,Z 777.52,A -85,B 0,C 180,E1 7112.131,E2 7112.131} C_VEL
LIN {X 0,Y 611.413,Z 766.372,A -85,B 0,C 180,E1 7117.84,E2 7117.84} C_VEL
LIN {X 0,Y 612.782,Z 740.706,A -85,B 0,C 180,E1 7123.598,E2 7123.598} C_VEL
LIN {X 0,Y 615.371,Z 701.505,A -85,B 0,C 180,E1 7128.815,E2 7128.815} C_VEL
LIN {X 0,Y 619.228,Z 651.161,A -85,B 0,C 180,E1 7133.079,E2 7133.079} C_VEL
LIN {X 0,Y 623.225,Z 591.742,A -85,B 0,C 180,E1 7136.17,E2 7136.17} C_VEL
LIN {X 0,Y 626.032,Z 530.382,A -85,B 0,C 180,E1 7137.828,E2 7137.828} C_VEL
LIN {X 0,Y 623.815,Z 507.178,A -85,B 0,C 180,E1 7138.271,E2 7138.271} C_VEL
LIN {X 0,Y 610.701,Z 474.78,A -85,B 0,C 180,E1 7139.539,E2 7139.539} C_VEL
LIN {X 0,Y 610.179,Z 474.78,A -85,B 0,C 180,E1 7148.372,E2 7148.372} C_VEL
LIN {X 0,Y 609.993,Z 474.78,A -85,B 0,C 180,E1 7157.171,E2 7157.171} C_VEL
LIN {X 0,Y 610.508,Z 474.78,A -85,B 0,C 180,E1 7165.951,E2 7165.951} C_VEL
LIN {X 0,Y 610.17,Z 474.78,A -85,B 0,C 180,E1 7175.115,E2 7175.115} C_VEL
LIN {X 0,Y 610.342,Z 474.78,A -85,B 0,C 180,E1 7183.345,E2 7183.345} C_VEL
LIN {X 0,Y 610.396,Z 474.78,A -85,B 0,C 180,E1 7192.099,E2 7192.099} C_VEL
LIN {X 0,Y 610.583,Z 474.78,A -85,B 0,C 180,E1 7199.245,E2 7199.245} C_VEL
LIN {X 0,Y 610.697,Z 474.78,A -85,B 0,C 180,E1 7206.376,E2 7206.376} C_VEL
LIN {X 0,Y 610.274,Z 474.78,A -85,B 0,C 180,E1 7215.088,E2 7215.088} C_VEL
LIN {X 0,Y 610.096,Z 474.78,A -85,B 0,C 180,E1 7222.626,E2 7222.626} C_VEL
LIN {X 0,Y 610.415,Z 474.78,A -85,B 0,C 180,E1 7231.007,E2 7231.007} C_VEL
LIN {X 0,Y 610.251,Z 474.78,A -85,B 0,C 180,E1 7239.29,E2 7239.29} C_VEL
LIN {X 0,Y 610.072,Z 474.78,A -85,B 0,C 180,E1 7247.13,E2 7247.13} C_VEL
LIN {X 0,Y 610.532,Z 474.78,A -85,B 0,C 180,E1 7256.022,E2 7256.022} C_VEL
LIN {X 0,Y 610.186,Z 474.78,A -85,B 0,C 180,E1 7265.069,E2 7265.069} C_VEL
LIN {X 0,Y 610.41,Z 474.78,A -85,B 0,C 180,E1 7273.399,E2 7273.399} C_VEL
LIN {X 0,Y 610.387,Z 474.78,A -85,B 0,C 180,E1 7282.146,E2 7282.146} C_VEL
LIN {X 0,Y 610.514,Z 474.78,A -85,B 0,C 180,E1 7289.288,E2 7289.288} C_VEL
LIN {X 0,Y 610.646,Z 474.78,A -85,B 0,C 180,E1 7296.416,E2 7296.416} C_VEL
LIN {X 0,Y 610.308,Z 474.78,A -85,B 0,C 180,E1 7305.124,E2 7305.124} C_VEL
LIN {X 0,Y 610.096,Z 474.78,A -85,B 0,C 180,E1 7312.661,E2 7312.661} C_VEL
LIN {X 0,Y 609.965,Z 474.78,A -85,B 0,C 180,E1 7320.974,E2 7320.974} C_VEL
LIN {X 0,Y 609.839,Z 474.78,A -85,B 0,C 180,E1 7329.354,E2 7329.354} C_VEL
LIN {X 0,Y 610.08,Z 474.78,A -85,B 0,C 180,E1 7337.163,E2 7337.163} C_VEL
LIN {X 0,Y 610.085,Z 474.78,A -85,B 0,C 180,E1 7346.378,E2 7346.378} C_VEL
LIN {X 0,Y 610.214,Z 474.78,A -85,B 0,C 180,E1 7355.106,E2 7355.106} C_VEL
LIN {X 0,Y 610.533,Z 474.78,A -85,B 0,C 180,E1 7363.439,E2 7363.439} C_VEL
LIN {X 0,Y 610.805,Z 474.78,A -85,B 0,C 180,E1 7370.752,E2 7370.752} C_VEL
LIN {X 0,Y 611.203,Z 474.78,A -85,B 0,C 180,E1 7377.909,E2 7377.909} C_VEL
LIN {X 0,Y 610.688,Z 474.78,A -85,B 0,C 180,E1 7386.462,E2 7386.462} C_VEL
LIN {X 0,Y 610.242,Z 474.78,A -85,B 0,C 180,E1 7395.177,E2 7395.177} C_VEL
LIN {X 0,Y 610.088,Z 474.78,A -85,B 0,C 180,E1 7402.719,E2 7402.719} C_VEL
LIN {X 0,Y 610.021,Z 474.78,A -85,B 0,C 180,E1 7410.945,E2 7410.945} C_VEL
LIN {X 0,Y 609.884,Z 474.78,A -85,B 0,C 180,E1 7419.428,E2 7419.428} C_VEL
LIN {X 0,Y 610.125,Z 474.78,A -85,B 0,C 180,E1 7427.251,E2 7427.251} C_VEL
LIN {X 0,Y 610.202,Z 474.78,A -85,B 0,C 180,E1 7431.859,E2 7431.859} C_VEL
LIN {X 0,Y 602.263,Z 474.78,A -85,B 0,C 180,E1 7435.136,E2 7435.136} C_VEL
LIN {X 0,Y 602.512,Z 475.027,A -85,B 0,C 180,E1 7440.21,E2 7440.21} C_VEL
LIN {X 0,Y 618.973,Z 521.011,A -85,B 0,C 180,E1 7441.68,E2 7441.68} C_VEL
LIN {X 0,Y 616.312,Z 585.67,A -85,B 0,C 180,E1 7443.268,E2 7443.268} C_VEL
LIN {X 0,Y 612.275,Z 644.742,A -85,B 0,C 180,E1 7446.198,E2 7446.198} C_VEL
LIN {X 0,Y 608.231,Z 695.549,A -85,B 0,C 180,E1 7450.331,E2 7450.331} C_VEL
LIN {X 0,Y 605.289,Z 735.765,A -85,B 0,C 180,E1 7455.434,E2 7455.434} C_VEL
LIN {X 0,Y 603.897,Z 763.762,A -85,B 0,C 180,E1 7461.334,E2 7461.334} C_VEL
LIN {X 0,Y 603.5,Z 775.79,A -85,B 0,C 180,E1 7466.398,E2 7466.398} C_VEL
LIN {X 0,Y 603.664,Z 777.345,A -85,B 0,C 180,E1 7472.159,E2 7472.159} C_VEL
LIN {X 0,Y 603.631,Z 765.02,A -85,B 0,C 180,E1 7478.306,E2 7478.306} C_VEL
LIN {X 0,Y 605.216,Z 737.724,A -85,B 0,C 180,E1 7484.258,E2 7484.258} C_VEL
LIN {X 0,Y 608.094,Z 697.428,A -85,B 0,C 180,E1 7489.484,E2 7489.484} C_VEL
LIN {X 0,Y 612.12,Z 646.256,A -85,B 0,C 180,E1 7493.701,E2 7493.701} C_VEL
LIN {X 0,Y 616.365,Z 586.493,A -85,B 0,C 180,E1 7496.695,E2 7496.695} C_VEL
LIN {X 0,Y 619.044,Z 523.088,A -85,B 0,C 180,E1 7498.284,E2 7498.284} C_VEL
LIN {X 0,Y 614.404,Z 503.425,A -85,B 0,C 180,E1 7498.79,E2 7498.79} C_VEL
LIN {X 0,Y 602.638,Z 474.78,A -85,B 0,C 180,E1 7499.944,E2 7499.944} C_VEL
LIN {X 0,Y 602.179,Z 474.78,A -85,B 0,C 180,E1 7508.097,E2 7508.097} C_VEL
LIN {X 0,Y 601.934,Z 474.78,A -85,B 0,C 180,E1 7516.06,E2 7516.06} C_VEL
LIN {X 0,Y 602.398,Z 474.78,A -85,B 0,C 180,E1 7524.901,E2 7524.901} C_VEL
LIN {X 0,Y 602.298,Z 474.78,A -85,B 0,C 180,E1 7533.795,E2 7533.795} C_VEL
LIN {X 0,Y 602.353,Z 474.78,A -85,B 0,C 180,E1 7543.117,E2 7543.117} C_VEL
LIN {X 0,Y 602.41,Z 474.78,A -85,B 0,C 180,E1 7551.994,E2 7551.994} C_VEL
LIN {X 0,Y 602.584,Z 474.78,A -85,B 0,C 180,E1 7559.235,E2 7559.235} C_VEL
LIN {X 0,Y 602.676,Z 474.78,A -85,B 0,C 180,E1 7566.461,E2 7566.461} C_VEL
LIN {X 0,Y 602.223,Z 474.78,A -85,B 0,C 180,E1 7575.294,E2 7575.294} C_VEL
LIN {X 0,Y 602.012,Z 474.78,A -85,B 0,C 180,E1 7583.155,E2 7583.155} C_VEL
LIN {X 0,Y 602.413,Z 474.78,A -85,B 0,C 180,E1 7591.034,E2 7591.034} C_VEL
LIN {X 0,Y 602.253,Z 474.78,A -85,B 0,C 180,E1 7599.915,E2 7599.915} C_VEL
LIN {X 0,Y 602.101,Z 474.78,A -85,B 0,C 180,E1 7608.13,E2 7608.13} C_VEL
LIN {X 0,Y 602.459,Z 474.78,A -85,B 0,C 180,E1 7615.503,E2 7615.503} C_VEL
LIN {X 0,Y 602.289,Z 474.78,A -85,B 0,C 180,E1 7623.856,E2 7623.856} C_VEL
LIN {X 0,Y 602.446,Z 474.78,A -85,B 0,C 180,E1 7633.173,E2 7633.173} C_VEL
LIN {X 0,Y 602.414,Z 474.78,A -85,B 0,C 180,E1 7642.042,E2 7642.042} C_VEL
LIN {X 0,Y 602.515,Z 474.78,A -85,B 0,C 180,E1 7649.279,E2 7649.279} C_VEL
LIN {X 0,Y 602.629,Z 474.78,A -85,B 0,C 180,E1 7656.502,E2 7656.502} C_VEL
LIN {X 0,Y 602.271,Z 474.78,A -85,B 0,C 180,E1 7665.33,E2 7665.33} C_VEL
LIN {X 0,Y 602.007,Z 474.78,A -85,B 0,C 180,E1 7673.199,E2 7673.199} C_VEL
LIN {X 0,Y 601.961,Z 474.78,A -85,B 0,C 180,E1 7681.094,E2 7681.094} C_VEL
LIN {X 0,Y 601.78,Z 474.78,A -85,B 0,C 180,E1 7689.986,E2 7689.986} C_VEL
LIN {X 0,Y 601.988,Z 474.78,A -85,B 0,C 180,E1 7698.154,E2 7698.154} C_VEL
LIN {X 0,Y 602.074,Z 474.78,A -85,B 0,C 180,E1 7707.245,E2 7707.245} C_VEL
LIN {X 0,Y 602.257,Z 474.78,A -85,B 0,C 180,E1 7715.486,E2 7715.486} C_VEL
LIN {X 0,Y 602.803,Z 474.78,A -85,B 0,C 180,E1 7724.721,E2 7724.721} C_VEL
LIN {X 0,Y 602.457,Z 474.78,A -85,B 0,C 180,E1 7732.082,E2 7732.082} C_VEL
LIN {X 0,Y 602.568,Z 474.78,A -85,B 0,C 180,E1 7739.322,E2 7739.322} C_VEL
LIN {X 0,Y 602.669,Z 474.78,A -85,B 0,C 180,E1 7746.548,E2 7746.548} C_VEL
LIN {X 0,Y 602.214,Z 474.78,A -85,B 0,C 180,E1 7755.384,E2 7755.384} C_VEL
LIN {X 0,Y 601.986,Z 474.78,A -85,B 0,C 180,E1 7763.149,E2 7763.149} C_VEL
LIN {X 0,Y 601.991,Z 474.78,A -85,B 0,C 180,E1 7771.159,E2 7771.159} C_VEL
LIN {X 0,Y 601.844,Z 474.78,A -85,B 0,C 180,E1 7780.06,E2 7780.06} C_VEL
LIN {X 0,Y 602.058,Z 474.78,A -85,B 0,C 180,E1 7788.126,E2 7788.126} C_VEL
LIN {X 0,Y 602.263,Z 474.78,A -85,B 0,C 180,E1 7795.136,E2 7795.136} C_VEL
LIN {X 0,Y 594.392,Z 474.78,A -85,B 0,C 180,E1 7798.447,E2 7798.447} C_VEL
LIN {X 0,Y 594.571,Z 476.022,A -85,B 0,C 180,E1 7799.787,E2 7799.787} C_VEL
LIN {X 0,Y 611.928,Z 523.298,A -85,B 0,C 180,E1 7801.364,E2 7801.364} C_VEL
LIN {X 0,Y 608.953,Z 587.845,A -85,B 0,C 180,E1 7803.018,E2 7803.018} C_VEL
LIN {X 0,Y 604.56,Z 647.573,A -85,B 0,C 180,E1 7806.093,E2 7806.093} C_VEL
LIN {X 0,Y 600.407,Z 697.249,A -85,B 0,C 180,E1 7810.256,E2 7810.256} C_VEL
LIN {X 0,Y 597.349,Z 737.009,A -85,B 0,C 180,E1 7815.464,E2 7815.464} C_VEL
LIN {X 0,Y 595.944,Z 763.586,A -85,B 0,C 180,E1 7821.218,E2 7821.218} C_VEL
LIN {X 0,Y 595.533,Z 775.615,A -85,B 0,C 180,E1 7826.35,E2 7826.35} C_VEL
LIN {X 0,Y 595.675,Z 777.17,A -85,B 0,C 180,E1 7832.188,E2 7832.188} C_VEL
LIN {X 0,Y 595.689,Z 764.844,A -85,B 0,C 180,E1 7838.417,E2 7838.417} C_VEL
LIN {X 0,Y 597.242,Z 738.716,A -85,B 0,C 180,E1 7844.258,E2 7844.258} C_VEL
LIN {X 0,Y 600.237,Z 698.955,A -85,B 0,C 180,E1 7849.558,E2 7849.558} C_VEL
LIN {X 0,Y 604.462,Z 648.343,A -85,B 0,C 180,E1 7853.855,E2 7853.855} C_VEL
LIN {X 0,Y 608.964,Z 589.03,A -85,B 0,C 180,E1 7856.931,E2 7856.931} C_VEL
LIN {X 0,Y 611.935,Z 525.57,A -85,B 0,C 180,E1 7858.599,E2 7858.599} C_VEL
LIN {X 0,Y 607.339,Z 505.496,A -85,B 0,C 180,E1 7859.127,E2 7859.127} C_VEL
LIN {X 0,Y 594.593,Z 474.78,A -85,B 0,C 180,E1 7860.261,E2 7860.261} C_VEL
LIN {X 0,Y 594.128,Z 474.78,A -85,B 0,C 180,E1 7868.773,E2 7868.773} C_VEL
LIN {X 0,Y 593.935,Z 474.78,A -85,B 0,C 180,E1 7877.335,E2 7877.335} C_VEL
LIN {X 0,Y 594.403,Z 474.78,A -85,B 0,C 180,E1 7886.013,E2 7886.013} C_VEL
LIN {X 0,Y 594.134,Z 474.78,A -85,B 0,C 180,E1 7895.032,E2 7895.032} C_VEL
LIN {X 0,Y 594.354,Z 474.78,A -85,B 0,C 180,E1 7903.099,E2 7903.099} C_VEL
LIN {X 0,Y 594.417,Z 474.78,A -85,B 0,C 180,E1 7911.886,E2 7911.886} C_VEL
LIN {X 0,Y 594.597,Z 474.78,A -85,B 0,C 180,E1 7919.225,E2 7919.225} C_VEL
LIN {X 0,Y 594.638,Z 474.78,A -85,B 0,C 180,E1 7926.549,E2 7926.549} C_VEL
LIN {X 0,Y 594.182,Z 474.78,A -85,B 0,C 180,E1 7935.506,E2 7935.506} C_VEL
LIN {X 0,Y 593.992,Z 474.78,A -85,B 0,C 180,E1 7943.275,E2 7943.275} C_VEL
LIN {X 0,Y 594.373,Z 474.78,A -85,B 0,C 180,E1 7951.502,E2 7951.502} C_VEL
LIN {X 0,Y 594.17,Z 474.78,A -85,B 0,C 180,E1 7960.57,E2 7960.57} C_VEL
LIN {X 0,Y 594.144,Z 474.78,A -85,B 0,C 180,E1 7969.394,E2 7969.394} C_VEL
LIN {X 0,Y 594.37,Z 474.78,A -85,B 0,C 180,E1 7976.732,E2 7976.732} C_VEL
LIN {X 0,Y 594.14,Z 474.78,A -85,B 0,C 180,E1 7985.093,E2 7985.093} C_VEL
LIN {X 0,Y 594.439,Z 474.78,A -85,B 0,C 180,E1 7993.012,E2 7993.012} C_VEL
LIN {X 0,Y 594.42,Z 474.78,A -85,B 0,C 180,E1 8001.934,E2 8001.934} C_VEL
LIN {X 0,Y 594.521,Z 474.78,A -85,B 0,C 180,E1 8009.269,E2 8009.269} C_VEL
LIN {X 0,Y 594.596,Z 474.78,A -85,B 0,C 180,E1 8016.59,E2 8016.59} C_VEL
LIN {X 0,Y 594.228,Z 474.78,A -85,B 0,C 180,E1 8025.543,E2 8025.543} C_VEL
LIN {X 0,Y 593.987,Z 474.78,A -85,B 0,C 180,E1 8033.311,E2 8033.311} C_VEL
LIN {X 0,Y 593.919,Z 474.78,A -85,B 0,C 180,E1 8041.563,E2 8041.563} C_VEL
LIN {X 0,Y 593.711,Z 474.78,A -85,B 0,C 180,E1 8050.642,E2 8050.642} C_VEL
LIN {X 0,Y 593.934,Z 474.78,A -85,B 0,C 180,E1 8059.41,E2 8059.41} C_VEL
LIN {X 0,Y 594.162,Z 474.78,A -85,B 0,C 180,E1 8068.763,E2 8068.763} C_VEL
LIN {X 0,Y 594.374,Z 474.78,A -85,B 0,C 180,E1 8078.323,E2 8078.323} C_VEL
LIN {X 0,Y 595.209,Z 474.78,A -85,B 0,C 180,E1 8087.531,E2 8087.531} C_VEL
LIN {X 0,Y 595.197,Z 474.78,A -85,B 0,C 180,E1 8097.852,E2 8097.852} C_VEL
LIN {X 0,Y 594.632,Z 474.78,A -85,B 0,C 180,E1 8106.637,E2 8106.637} C_VEL
LIN {X 0,Y 594.172,Z 474.78,A -85,B 0,C 180,E1 8115.598,E2 8115.598} C_VEL
LIN {X 0,Y 593.958,Z 474.78,A -85,B 0,C 180,E1 8123.372,E2 8123.372} C_VEL
LIN {X 0,Y 593.953,Z 474.78,A -85,B 0,C 180,E1 8131.629,E2 8131.629} C_VEL
LIN {X 0,Y 593.79,Z 474.78,A -85,B 0,C 180,E1 8140.717,E2 8140.717} C_VEL
LIN {X 0,Y 594.033,Z 474.78,A -85,B 0,C 180,E1 8149.384,E2 8149.384} C_VEL
